RoboDK station: irb120.rdk

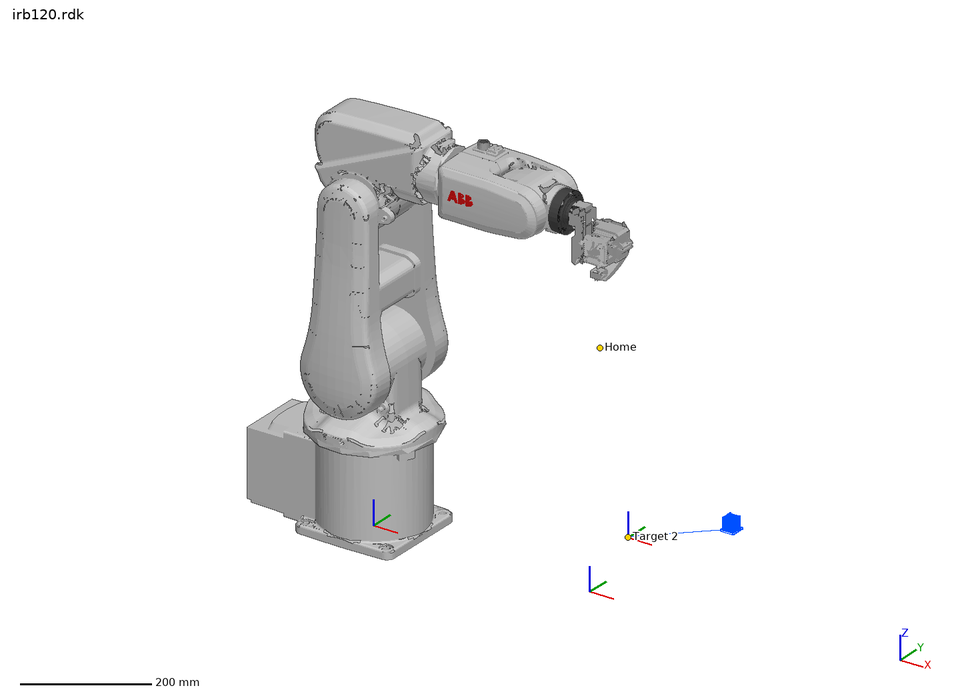
[picture v0: the station drawn from its stored meshes, robots at their saved joint values, targets as dots, program paths as lines]
Station irb120_V12 (saved by RoboDK 5.2.5). Poses are relative to the parent item; angles as X-Y-Z fixed-axis rotations.
  - frame ABB IRB 120-3/0.6 Base at (-494.33, 30.55, 0) mm
    - robot ABB IRB 120-3/0.6: 6 axes, payload 3 kg, reach 580 mm, repeatability 0.01 mm, weight 25 kg
        modified DH rows (alpha deg, a mm, theta deg, d mm): 0, 0, 0, 290; -90, 0, -90, 0; 0, 270, 0, 0; -90, 70, 0, 302; 90, 0, 0, 0; -90, 0, 180, 72
        joint limits [-165, -110, -90, -160, -120, -400] to [165, 110, 70, 160, 120, 400]; home [0, 0, 0, 0, 0, 0]; saved at [0, 0, 0, 0, 0, 0]
      - tool EndEffector, TCP at (101, 0, 38) mm, rotated rx 0 ry 90 rz 0 deg, size 98.6 x 123.3 x 80.9 mm, geometry from EndEffector.stl
  - frame Robot Table at (-94.33, 30.55, 0) mm
    - object Table at (0, 0, 0) mm, size 926 x 772 x 180 mm, geometry from Table.stl
  - frame Print at (40, -60, 165.5) mm
    - target Home (joint target) at (16.67, -99.45, 364) mm, rotated rx -180 ry 0 rz -180 deg; joints [0, 0, 0, 0, 0, 0] of ABB IRB 120-3/0.6
    - target Target 2 (Cartesian target) at (0, 0, 0) mm, rotated rx 180 ry 0 rz 180 deg; joints [-12.046, 47.993, 6.255, -14.732, -55.151, 8.545] of ABB IRB 120-3/0.6
  - Python program Prog2 (listed below)
  - camera Camera 1
  - frame Frame 4 at (1070.92, -4.45, 581.3) mm, rotated rx -103 ry 0 rz 90 deg
  - program out (41618 instructions, listed below)
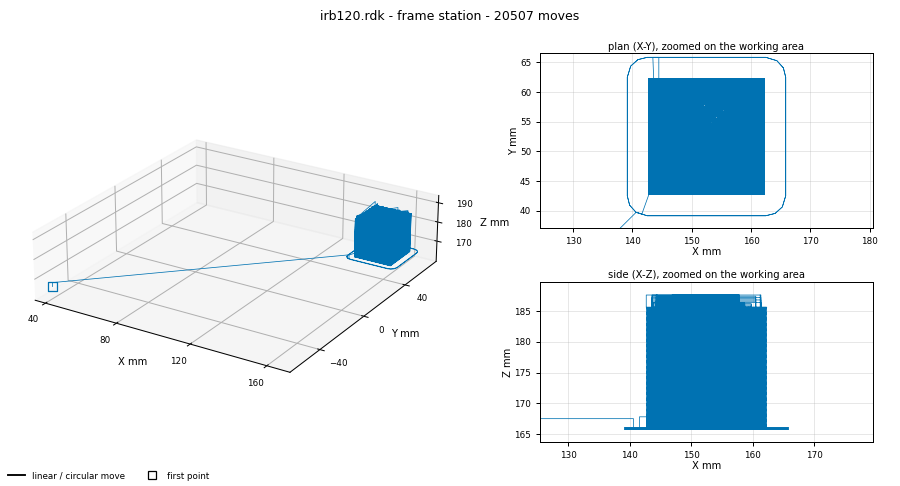
[picture p0: tool path of irb120.rdk in frame station, 20507 of 20507 moves have a stored position in this frame; points joined in program order, loops and branches not executed]

--- Python program Prog2 ---
# Type help("robolink") or help("robodk") for more information
# Press F5 to run the script
# Documentation: https://robodk.com/doc/en/RoboDK-API.html
# Reference:     https://robodk.com/doc/en/PythonAPI/index.html
# Note: It is not required to keep a copy of this file, your python script is saved with the station
from robolink import *    # RoboDK API
from robodk import *      # Robot toolbox
RDK = Robolink()
import cv2
import tempfile
import numpy as np
import math
# # Notify user:
# print('To edit this program:\nright click on the Python program, then, select "Edit Python script"')

# RDK = Robolink() # connect to the RoboDK API (RoboDK starts if it has not started)
# robot  = RDK.Item('', ITEM_TYPE_ROBOT)   # Retrieve the robot
# joints = robot.Joints().list()          # retrieve the current robot joints as a list
# joints[5] = 20                           # set joint 6 to 0 deg
# robot.MoveJ(joints)
# s=robot.JointPoses()
# Print("finish")
CAM_NAME = "Camera 1"
cam_item = RDK.Item(CAM_NAME, ITEM_TYPE_CAMERA)
if not cam_item.Valid():
    raise Exception("Camera not found! %s" % CAM_NAME)

tempdir = tempfile.gettempdir()
snapshot_file = tempdir + "\\sift_temp.png"
print(snapshot_file)
imgdir="C:/Users/dell/Desktop/RoboDk/Robotirb120/00006000.jpg"
image = cv2.imread(imgdir)
image=cv2.resize(image,(640,480))
while(1):
    RDK.Cam2D_Snapshot(snapshot_file, cam_item)
    img_scene = cv2.imread(snapshot_file, cv2.IMREAD_GRAYSCALE)
    img_scene=cv2.resize(img_scene,(640,480))
    (thresh, im_bw) = cv2.threshold(img_scene, 128, 255, cv2.THRESH_BINARY | cv2.THRESH_OTSU)
    # print(image.shape)
    # print(im_bw.shape)
    kernel = np.ones((3,3),np.uint8)
    closing = cv2.morphologyEx(im_bw, cv2.MORPH_CLOSE, kernel)
    gradient = cv2.morphologyEx(im_bw, cv2.MORPH_GRADIENT, kernel)
    masked = cv2.bitwise_and(image, image, mask=closing)
    vis = np.concatenate((image,masked), axis=1)
    cv2.imshow("image3",masked)
    key = cv2.waitKey(1)
    if key == 27:
        break  # User pressed ESC, exit

--- program out (robot ABB IRB 120-3/0.6) ---
  Set Ref.: Print
  Set Tool at (101, 0, 38) mm, rotated rx 0 ry 90 rz 0 deg
  Smooth(2)
  Set accel. (1000.0 mm/s2)
  Call Mcode M107
  MoveJ (T0) to (0, 0, 0) mm, rotated rx 180 ry 0 rz -180 deg; joints [0, 0, 0, 0, 0, 0]
  Call Mcode M190 S50
  MoveL (T1) to (0, 0, 0) mm, rotated rx 180 ry 0 rz -180 deg; joints [0, 0, 0, 0, 0, 0]
  Call Mcode M104 S200
  MoveL (T2) to (0, 0, 0) mm, rotated rx 180 ry 0 rz -180 deg; joints [0, 0, 0, 0, 0, 0]
  Call Mcode M109 S200
  MoveL (T3) to (0, 0, 0) mm, rotated rx 180 ry 0 rz -180 deg; joints [0, 0, 0, 0, 0, 0]
  Call Mcode M83
  MoveL (T4) to (0, 0, 0) mm, rotated rx 180 ry 0 rz -180 deg; joints [0, 0, 0, 0, 0, 0]
  Call Mcode M107
  MoveL (T5) to (0, 0, 0) mm, rotated rx 180 ry 0 rz -180 deg; joints [0, 0, 0, 0, 0, 0]
  Set speed (45.0 mm/s)
  Call Extruder -2.0
  MoveL (T6) to (0, 0, 0) mm, rotated rx 180 ry 0 rz -180 deg; joints [0, 0, 0, 0, 0, 0]
  Set speed (150.0 mm/s)
  MoveL (T7) to (0, 0, 2) mm, rotated rx 180 ry 0 rz -180 deg; joints [0, 0, 0, 0, 0, 0]
  MoveL (T8) to (100.63, 99.72, 2) mm, rotated rx 180 ry 0 rz -180 deg; joints [0, 0, 0, 0, 0, 0]
  MoveL (T9) to (100.63, 99.72, 0.3) mm, rotated rx 180 ry 0 rz -180 deg; joints [0, 0, 0, 0, 0, 0]
  Set speed (40.0 mm/s)
  Call Extruder 2.0
  MoveL (T10) to (100.63, 99.72, 0.3) mm, rotated rx 180 ry 0 rz -180 deg; joints [0, 0, 0, 0, 0, 0]
  Call Extruder 2.0
  Call Mcode M204 P1000
  MoveL (T11) to (100.63, 99.72, 0.3) mm, rotated rx 180 ry 0 rz -180 deg; joints [0, 0, 0, 0, 0, 0]
  Set speed (20.0 mm/s)
  MoveL (T12) to (100.63, 99.72, 0.3) mm, rotated rx 180 ry 0 rz -180 deg; joints [0, 0, 0, 0, 0, 0]
  Call Extruder 0.07812
  MoveL (T13) to (102.5, 99.14, 0.3) mm, rotated rx 180 ry 0 rz -180 deg; joints [0, 0, 0, 0, 0, 0]
  Call Extruder 0.79839
  MoveL (T14) to (122.5, 99.14, 0.3) mm, rotated rx 180 ry 0 rz -180 deg; joints [0, 0, 0, 0, 0, 0]
  Call Extruder 0.06492
  MoveL (T15) to (124.08, 99.54, 0.3) mm, rotated rx 180 ry 0 rz -180 deg; joints [0, 0, 0, 0, 0, 0]
  Call Extruder 0.06492
  MoveL (T16) to (125.28, 100.63, 0.3) mm, rotated rx 180 ry 0 rz -180 deg; joints [0, 0, 0, 0, 0, 0]
  Call Extruder 0.07812
  MoveL (T17) to (125.86, 102.5, 0.3) mm, rotated rx 180 ry 0 rz -180 deg; joints [0, 0, 0, 0, 0, 0]
  Call Extruder 0.79839
  MoveL (T18) to (125.86, 122.5, 0.3) mm, rotated rx 180 ry 0 rz -180 deg; joints [0, 0, 0, 0, 0, 0]
  Call Extruder 0.06492
  MoveL (T19) to (125.46, 124.08, 0.3) mm, rotated rx 180 ry 0 rz -180 deg; joints [0, 0, 0, 0, 0, 0]
  Call Extruder 0.06492
  MoveL (T20) to (124.37, 125.28, 0.3) mm, rotated rx 180 ry 0 rz -180 deg; joints [0, 0, 0, 0, 0, 0]
  Call Extruder 0.07812
  MoveL (T21) to (122.5, 125.86, 0.3) mm, rotated rx 180 ry 0 rz -180 deg; joints [0, 0, 0, 0, 0, 0]
  Call Extruder 0.79839
  MoveL (T22) to (102.5, 125.86, 0.3) mm, rotated rx 180 ry 0 rz -180 deg; joints [0, 0, 0, 0, 0, 0]
  Call Extruder 0.06492
  MoveL (T23) to (100.92, 125.46, 0.3) mm, rotated rx 180 ry 0 rz -180 deg; joints [0, 0, 0, 0, 0, 0]
  Call Extruder 0.06492
  MoveL (T24) to (99.72, 124.37, 0.3) mm, rotated rx 180 ry 0 rz -180 deg; joints [0, 0, 0, 0, 0, 0]
  Call Extruder 0.07812
  MoveL (T25) to (99.14, 122.5, 0.3) mm, rotated rx 180 ry 0 rz -180 deg; joints [0, 0, 0, 0, 0, 0]
  Call Extruder 0.79839
  MoveL (T26) to (99.14, 102.5, 0.3) mm, rotated rx 180 ry 0 rz -180 deg; joints [0, 0, 0, 0, 0, 0]
  Call Extruder 0.06492
  MoveL (T27) to (99.54, 100.92, 0.3) mm, rotated rx 180 ry 0 rz -180 deg; joints [0, 0, 0, 0, 0, 0]
  Call Extruder 0.06252
  MoveL (T28) to (100.59, 99.76, 0.3) mm, rotated rx 180 ry 0 rz -180 deg; joints [0, 0, 0, 0, 0, 0]
  Set speed (45.0 mm/s)
  Call Extruder -1.6
  MoveL (T29) to (100.59, 99.76, 0.3) mm, rotated rx 180 ry 0 rz -180 deg; joints [0, 0, 0, 0, 0, 0]
  Set speed (120.0 mm/s)
  MoveL (T30) to (100.59, 99.76, 0.3) mm, rotated rx 180 ry 0 rz -180 deg; joints [0, 0, 0, 0, 0, 0]
  Call Extruder -0.38
  MoveL (T31) to (101.6, 99.43, 0.3) mm, rotated rx 180 ry 0 rz -180 deg; joints [0, 0, 0, 0, 0, 0]
  Set speed (45.0 mm/s)
  Call Extruder -0.02
  MoveL (T32) to (101.6, 99.43, 0.3) mm, rotated rx 180 ry 0 rz -180 deg; joints [0, 0, 0, 0, 0, 0]
  Set speed (150.0 mm/s)
  MoveL (T33) to (101.6, 99.43, 2.3) mm, rotated rx 180 ry 0 rz -180 deg; joints [0, 0, 0, 0, 0, 0]
  MoveL (T34) to (102.81, 102.81, 2.3) mm, rotated rx 180 ry 0 rz -180 deg; joints [0, 0, 0, 0, 0, 0]
  MoveL (T35) to (102.81, 102.81, 0.3) mm, rotated rx 180 ry 0 rz -180 deg; joints [0, 0, 0, 0, 0, 0]
  Set speed (40.0 mm/s)
  Call Extruder 2.0
  MoveL (T36) to (102.81, 102.81, 0.3) mm, rotated rx 180 ry 0 rz -180 deg; joints [0, 0, 0, 0, 0, 0]
  Set speed (20.0 mm/s)
  MoveL (T37) to (102.81, 102.81, 0.3) mm, rotated rx 180 ry 0 rz -180 deg; joints [0, 0, 0, 0, 0, 0]
  Call Extruder 0.77364
  MoveL (T38) to (122.19, 102.81, 0.3) mm, rotated rx 180 ry 0 rz -180 deg; joints [0, 0, 0, 0, 0, 0]
  Call Extruder 0.77364
  MoveL (T39) to (122.19, 122.19, 0.3) mm, rotated rx 180 ry 0 rz -180 deg; joints [0, 0, 0, 0, 0, 0]
  Call Extruder 0.77364
  MoveL (T40) to (102.81, 122.19, 0.3) mm, rotated rx 180 ry 0 rz -180 deg; joints [0, 0, 0, 0, 0, 0]
  Call Extruder 0.77124
  MoveL (T41) to (102.81, 102.87, 0.3) mm, rotated rx 180 ry 0 rz -180 deg; joints [0, 0, 0, 0, 0, 0]
  Set speed (150.0 mm/s)
  MoveL (T42) to (103.2, 102.91, 0.3) mm, rotated rx 180 ry 0 rz -180 deg; joints [0, 0, 0, 0, 0, 0]
  Set speed (45.0 mm/s)
  Call Extruder -1.6
  MoveL (T43) to (103.2, 102.91, 0.3) mm, rotated rx 180 ry 0 rz -180 deg; joints [0, 0, 0, 0, 0, 0]
  Set speed (120.0 mm/s)
  MoveL (T44) to (103.2, 102.91, 0.3) mm, rotated rx 180 ry 0 rz -180 deg; joints [0, 0, 0, 0, 0, 0]
  Call Extruder -0.38
  MoveL (T45) to (103.88, 102.87, 0.3) mm, rotated rx 180 ry 0 rz -180 deg; joints [0, 0, 0, 0, 0, 0]
  Set speed (45.0 mm/s)
  Call Extruder -0.02
  MoveL (T46) to (103.88, 102.87, 0.3) mm, rotated rx 180 ry 0 rz -180 deg; joints [0, 0, 0, 0, 0, 0]
  Set speed (150.0 mm/s)
  MoveL (T47) to (103.88, 102.87, 2.3) mm, rotated rx 180 ry 0 rz -180 deg; joints [0, 0, 0, 0, 0, 0]
  MoveL (T48) to (121.83, 121.83, 2.3) mm, rotated rx 180 ry 0 rz -180 deg; joints [0, 0, 0, 0, 0, 0]
  MoveL (T49) to (121.83, 121.83, 0.3) mm, rotated rx 180 ry 0 rz -180 deg; joints [0, 0, 0, 0, 0, 0]
  Set speed (40.0 mm/s)
  Call Extruder 2.0
  MoveL (T50) to (121.83, 121.83, 0.3) mm, rotated rx 180 ry 0 rz -180 deg; joints [0, 0, 0, 0, 0, 0]
  Set speed (20.0 mm/s)
  MoveL (T51) to (121.83, 121.83, 0.3) mm, rotated rx 180 ry 0 rz -180 deg; joints [0, 0, 0, 0, 0, 0]
  Call Extruder 0.74524
  MoveL (T52) to (103.17, 121.83, 0.3) mm, rotated rx 180 ry 0 rz -180 deg; joints [0, 0, 0, 0, 0, 0]
  Call Extruder 0.74524
  MoveL (T53) to (103.17, 103.17, 0.3) mm, rotated rx 180 ry 0 rz -180 deg; joints [0, 0, 0, 0, 0, 0]
  Call Extruder 0.74524
  MoveL (T54) to (121.83, 103.17, 0.3) mm, rotated rx 180 ry 0 rz -180 deg; joints [0, 0, 0, 0, 0, 0]
  Call Extruder 0.74285
  MoveL (T55) to (121.83, 121.77, 0.3) mm, rotated rx 180 ry 0 rz -180 deg; joints [0, 0, 0, 0, 0, 0]
  Set speed (150.0 mm/s)
  MoveL (T56) to (121.48, 121.48, 0.3) mm, rotated rx 180 ry 0 rz -180 deg; joints [0, 0, 0, 0, 0, 0]
  Set speed (20.0 mm/s)
  MoveL (T57) to (121.48, 121.48, 0.3) mm, rotated rx 180 ry 0 rz -180 deg; joints [0, 0, 0, 0, 0, 0]
  Call Extruder 0.71685
  MoveL (T58) to (103.52, 121.48, 0.3) mm, rotated rx 180 ry 0 rz -180 deg; joints [0, 0, 0, 0, 0, 0]
  Call Extruder 0.71685
  MoveL (T59) to (103.52, 103.52, 0.3) mm, rotated rx 180 ry 0 rz -180 deg; joints [0, 0, 0, 0, 0, 0]
  Call Extruder 0.71685
  MoveL (T60) to (121.48, 103.52, 0.3) mm, rotated rx 180 ry 0 rz -180 deg; joints [0, 0, 0, 0, 0, 0]
  Call Extruder 0.71446
  MoveL (T61) to (121.48, 121.42, 0.3) mm, rotated rx 180 ry 0 rz -180 deg; joints [0, 0, 0, 0, 0, 0]
  Set speed (45.0 mm/s)
  Call Extruder -1.6
  MoveL (T62) to (121.48, 121.42, 0.3) mm, rotated rx 180 ry 0 rz -180 deg; joints [0, 0, 0, 0, 0, 0]
  Set speed (120.0 mm/s)
  MoveL (T63) to (121.48, 121.42, 0.3) mm, rotated rx 180 ry 0 rz -180 deg; joints [0, 0, 0, 0, 0, 0]
  Call Extruder -0.38
  MoveL (T64) to (120.41, 121.42, 0.3) mm, rotated rx 180 ry 0 rz -180 deg; joints [0, 0, 0, 0, 0, 0]
  Set speed (45.0 mm/s)
  Call Extruder -0.02
  MoveL (T65) to (120.41, 121.42, 0.3) mm, rotated rx 180 ry 0 rz -180 deg; joints [0, 0, 0, 0, 0, 0]
  Set speed (150.0 mm/s)
  MoveL (T66) to (120.41, 121.42, 2.3) mm, rotated rx 180 ry 0 rz -180 deg; joints [0, 0, 0, 0, 0, 0]
  MoveL (T67) to (120.65, 103.63, 2.3) mm, rotated rx 180 ry 0 rz -180 deg; joints [0, 0, 0, 0, 0, 0]
  MoveL (T68) to (120.65, 103.63, 0.3) mm, rotated rx 180 ry 0 rz -180 deg; joints [0, 0, 0, 0, 0, 0]
  Set speed (40.0 mm/s)
  Call Extruder 2.0
  MoveL (T69) to (120.65, 103.63, 0.3) mm, rotated rx 180 ry 0 rz -180 deg; joints [0, 0, 0, 0, 0, 0]
  Set speed (20.0 mm/s)
  MoveL (T70) to (120.65, 103.63, 0.3) mm, rotated rx 180 ry 0 rz -180 deg; joints [0, 0, 0, 0, 0, 0]
  Call Extruder 0.0323
  MoveL (T71) to (121.21, 104.19, 0.3) mm, rotated rx 180 ry 0 rz -180 deg; joints [0, 0, 0, 0, 0, 0]
  Call Extruder 0.02048
  MoveL (T72) to (121.21, 104.7, 0.3) mm, rotated rx 180 ry 0 rz -180 deg; joints [0, 0, 0, 0, 0, 0]
  Call Extruder 0.05214
  MoveL (T73) to (120.3, 103.79, 0.3) mm, rotated rx 180 ry 0 rz -180 deg; joints [0, 0, 0, 0, 0, 0]
  Call Extruder 0.02048
  MoveL (T74) to (119.79, 103.79, 0.3) mm, rotated rx 180 ry 0 rz -180 deg; joints [0, 0, 0, 0, 0, 0]
  Call Extruder 0.08111
  MoveL (T75) to (121.21, 105.21, 0.3) mm, rotated rx 180 ry 0 rz -180 deg; joints [0, 0, 0, 0, 0, 0]
  Call Extruder 0.02048
  MoveL (T76) to (121.21, 105.72, 0.3) mm, rotated rx 180 ry 0 rz -180 deg; joints [0, 0, 0, 0, 0, 0]
  Call Extruder 0.11008
  MoveL (T77) to (119.28, 103.79, 0.3) mm, rotated rx 180 ry 0 rz -180 deg; joints [0, 0, 0, 0, 0, 0]
  Call Extruder 0.02048
  MoveL (T78) to (118.77, 103.79, 0.3) mm, rotated rx 180 ry 0 rz -180 deg; joints [0, 0, 0, 0, 0, 0]
  Call Extruder 0.13905
  MoveL (T79) to (121.21, 106.23, 0.3) mm, rotated rx 180 ry 0 rz -180 deg; joints [0, 0, 0, 0, 0, 0]
  Call Extruder 0.02048
  MoveL (T80) to (121.21, 106.73, 0.3) mm, rotated rx 180 ry 0 rz -180 deg; joints [0, 0, 0, 0, 0, 0]
  Call Extruder 0.16801
  MoveL (T81) to (118.27, 103.79, 0.3) mm, rotated rx 180 ry 0 rz -180 deg; joints [0, 0, 0, 0, 0, 0]
  Call Extruder 0.02048
  MoveL (T82) to (117.76, 103.79, 0.3) mm, rotated rx 180 ry 0 rz -180 deg; joints [0, 0, 0, 0, 0, 0]
  Call Extruder 0.19698
  MoveL (T83) to (121.21, 107.24, 0.3) mm, rotated rx 180 ry 0 rz -180 deg; joints [0, 0, 0, 0, 0, 0]
  Call Extruder 0.02048
  MoveL (T84) to (121.21, 107.75, 0.3) mm, rotated rx 180 ry 0 rz -180 deg; joints [0, 0, 0, 0, 0, 0]
  Call Extruder 0.22595
  MoveL (T85) to (117.25, 103.79, 0.3) mm, rotated rx 180 ry 0 rz -180 deg; joints [0, 0, 0, 0, 0, 0]
  Call Extruder 0.02048
  MoveL (T86) to (116.74, 103.79, 0.3) mm, rotated rx 180 ry 0 rz -180 deg; joints [0, 0, 0, 0, 0, 0]
  Call Extruder 0.25492
  MoveL (T87) to (121.21, 108.26, 0.3) mm, rotated rx 180 ry 0 rz -180 deg; joints [0, 0, 0, 0, 0, 0]
  Call Extruder 0.02048
  MoveL (T88) to (121.21, 108.77, 0.3) mm, rotated rx 180 ry 0 rz -180 deg; joints [0, 0, 0, 0, 0, 0]
  Call Extruder 0.28388
  MoveL (T89) to (116.23, 103.79, 0.3) mm, rotated rx 180 ry 0 rz -180 deg; joints [0, 0, 0, 0, 0, 0]
  Call Extruder 0.02048
  MoveL (T90) to (115.73, 103.79, 0.3) mm, rotated rx 180 ry 0 rz -180 deg; joints [0, 0, 0, 0, 0, 0]
  Call Extruder 0.31285
  MoveL (T91) to (121.21, 109.27, 0.3) mm, rotated rx 180 ry 0 rz -180 deg; joints [0, 0, 0, 0, 0, 0]
  Call Extruder 0.02048
  MoveL (T92) to (121.21, 109.78, 0.3) mm, rotated rx 180 ry 0 rz -180 deg; joints [0, 0, 0, 0, 0, 0]
  Call Extruder 0.34182
  MoveL (T93) to (115.22, 103.79, 0.3) mm, rotated rx 180 ry 0 rz -180 deg; joints [0, 0, 0, 0, 0, 0]
  Call Extruder 0.02048
  MoveL (T94) to (114.71, 103.79, 0.3) mm, rotated rx 180 ry 0 rz -180 deg; joints [0, 0, 0, 0, 0, 0]
  Call Extruder 0.37079
  MoveL (T95) to (121.21, 110.29, 0.3) mm, rotated rx 180 ry 0 rz -180 deg; joints [0, 0, 0, 0, 0, 0]
  Call Extruder 0.02048
  MoveL (T96) to (121.21, 110.8, 0.3) mm, rotated rx 180 ry 0 rz -180 deg; joints [0, 0, 0, 0, 0, 0]
  Call Extruder 0.39975
  MoveL (T97) to (114.2, 103.79, 0.3) mm, rotated rx 180 ry 0 rz -180 deg; joints [0, 0, 0, 0, 0, 0]
  Call Extruder 0.02048
  MoveL (T98) to (113.69, 103.79, 0.3) mm, rotated rx 180 ry 0 rz -180 deg; joints [0, 0, 0, 0, 0, 0]
  Call Extruder 0.42872
  MoveL (T99) to (121.21, 111.31, 0.3) mm, rotated rx 180 ry 0 rz -180 deg; joints [0, 0, 0, 0, 0, 0]
  Call Extruder 0.02048
  MoveL (T100) to (121.21, 111.81, 0.3) mm, rotated rx 180 ry 0 rz -180 deg; joints [0, 0, 0, 0, 0, 0]
  Call Extruder 0.45769
  MoveL (T101) to (113.19, 103.79, 0.3) mm, rotated rx 180 ry 0 rz -180 deg; joints [0, 0, 0, 0, 0, 0]
  Call Extruder 0.02048
  MoveL (T102) to (112.68, 103.79, 0.3) mm, rotated rx 180 ry 0 rz -180 deg; joints [0, 0, 0, 0, 0, 0]
  Call Extruder 0.48666
  MoveL (T103) to (121.21, 112.32, 0.3) mm, rotated rx 180 ry 0 rz -180 deg; joints [0, 0, 0, 0, 0, 0]
  Call Extruder 0.02048
  MoveL (T104) to (121.21, 112.83, 0.3) mm, rotated rx 180 ry 0 rz -180 deg; joints [0, 0, 0, 0, 0, 0]
  Call Extruder 0.51562
  MoveL (T105) to (112.17, 103.79, 0.3) mm, rotated rx 180 ry 0 rz -180 deg; joints [0, 0, 0, 0, 0, 0]
  Call Extruder 0.02048
  MoveL (T106) to (111.66, 103.79, 0.3) mm, rotated rx 180 ry 0 rz -180 deg; joints [0, 0, 0, 0, 0, 0]
  Call Extruder 0.54459
  MoveL (T107) to (121.21, 113.34, 0.3) mm, rotated rx 180 ry 0 rz -180 deg; joints [0, 0, 0, 0, 0, 0]
  Call Extruder 0.02048
  MoveL (T108) to (121.21, 113.85, 0.3) mm, rotated rx 180 ry 0 rz -180 deg; joints [0, 0, 0, 0, 0, 0]
  Call Extruder 0.57356
  MoveL (T109) to (111.15, 103.79, 0.3) mm, rotated rx 180 ry 0 rz -180 deg; joints [0, 0, 0, 0, 0, 0]
  Call Extruder 0.02048
  MoveL (T110) to (110.65, 103.79, 0.3) mm, rotated rx 180 ry 0 rz -180 deg; joints [0, 0, 0, 0, 0, 0]
  Call Extruder 0.60253
  MoveL (T111) to (121.21, 114.35, 0.3) mm, rotated rx 180 ry 0 rz -180 deg; joints [0, 0, 0, 0, 0, 0]
  Call Extruder 0.02048
  MoveL (T112) to (121.21, 114.86, 0.3) mm, rotated rx 180 ry 0 rz -180 deg; joints [0, 0, 0, 0, 0, 0]
  Call Extruder 0.63149
  MoveL (T113) to (110.14, 103.79, 0.3) mm, rotated rx 180 ry 0 rz -180 deg; joints [0, 0, 0, 0, 0, 0]
  Call Extruder 0.02048
  MoveL (T114) to (109.63, 103.79, 0.3) mm, rotated rx 180 ry 0 rz -180 deg; joints [0, 0, 0, 0, 0, 0]
  Call Extruder 0.66046
  MoveL (T115) to (121.21, 115.37, 0.3) mm, rotated rx 180 ry 0 rz -180 deg; joints [0, 0, 0, 0, 0, 0]
  Call Extruder 0.02048
  MoveL (T116) to (121.21, 115.88, 0.3) mm, rotated rx 180 ry 0 rz -180 deg; joints [0, 0, 0, 0, 0, 0]
  Call Extruder 0.68943
  MoveL (T117) to (109.12, 103.79, 0.3) mm, rotated rx 180 ry 0 rz -180 deg; joints [0, 0, 0, 0, 0, 0]
  Call Extruder 0.02048
  MoveL (T118) to (108.61, 103.79, 0.3) mm, rotated rx 180 ry 0 rz -180 deg; joints [0, 0, 0, 0, 0, 0]
  Call Extruder 0.7184
  MoveL (T119) to (121.21, 116.39, 0.3) mm, rotated rx 180 ry 0 rz -180 deg; joints [0, 0, 0, 0, 0, 0]
  Call Extruder 0.02048
  MoveL (T120) to (121.21, 116.89, 0.3) mm, rotated rx 180 ry 0 rz -180 deg; joints [0, 0, 0, 0, 0, 0]
  Call Extruder 0.74736
  MoveL (T121) to (108.11, 103.79, 0.3) mm, rotated rx 180 ry 0 rz -180 deg; joints [0, 0, 0, 0, 0, 0]
  Call Extruder 0.02048
  MoveL (T122) to (107.6, 103.79, 0.3) mm, rotated rx 180 ry 0 rz -180 deg; joints [0, 0, 0, 0, 0, 0]
  Call Extruder 0.77633
  MoveL (T123) to (121.21, 117.4, 0.3) mm, rotated rx 180 ry 0 rz -180 deg; joints [0, 0, 0, 0, 0, 0]
  Call Extruder 0.02048
  MoveL (T124) to (121.21, 117.91, 0.3) mm, rotated rx 180 ry 0 rz -180 deg; joints [0, 0, 0, 0, 0, 0]
  Call Extruder 0.8053
  MoveL (T125) to (107.09, 103.79, 0.3) mm, rotated rx 180 ry 0 rz -180 deg; joints [0, 0, 0, 0, 0, 0]
  Call Extruder 0.02048
  MoveL (T126) to (106.58, 103.79, 0.3) mm, rotated rx 180 ry 0 rz -180 deg; joints [0, 0, 0, 0, 0, 0]
  Call Extruder 0.83426
  MoveL (T127) to (121.21, 118.42, 0.3) mm, rotated rx 180 ry 0 rz -180 deg; joints [0, 0, 0, 0, 0, 0]
  Call Extruder 0.02048
  MoveL (T128) to (121.21, 118.93, 0.3) mm, rotated rx 180 ry 0 rz -180 deg; joints [0, 0, 0, 0, 0, 0]
  Call Extruder 0.86323
  MoveL (T129) to (106.07, 103.79, 0.3) mm, rotated rx 180 ry 0 rz -180 deg; joints [0, 0, 0, 0, 0, 0]
  Call Extruder 0.02048
  MoveL (T130) to (105.57, 103.79, 0.3) mm, rotated rx 180 ry 0 rz -180 deg; joints [0, 0, 0, 0, 0, 0]
  Call Extruder 0.8922
  MoveL (T131) to (121.21, 119.43, 0.3) mm, rotated rx 180 ry 0 rz -180 deg; joints [0, 0, 0, 0, 0, 0]
  Call Extruder 0.02048
  MoveL (T132) to (121.21, 119.94, 0.3) mm, rotated rx 180 ry 0 rz -180 deg; joints [0, 0, 0, 0, 0, 0]
  Call Extruder 0.92117
  MoveL (T133) to (105.06, 103.79, 0.3) mm, rotated rx 180 ry 0 rz -180 deg; joints [0, 0, 0, 0, 0, 0]
  Call Extruder 0.02048
  MoveL (T134) to (104.55, 103.79, 0.3) mm, rotated rx 180 ry 0 rz -180 deg; joints [0, 0, 0, 0, 0, 0]
  Call Extruder 0.95013
  MoveL (T135) to (121.21, 120.45, 0.3) mm, rotated rx 180 ry 0 rz -180 deg; joints [0, 0, 0, 0, 0, 0]
  Call Extruder 0.02048
  MoveL (T136) to (121.21, 120.96, 0.3) mm, rotated rx 180 ry 0 rz -180 deg; joints [0, 0, 0, 0, 0, 0]
  Call Extruder 0.9791
  MoveL (T137) to (104.04, 103.79, 0.3) mm, rotated rx 180 ry 0 rz -180 deg; joints [0, 0, 0, 0, 0, 0]
  Call Extruder 0.01024
  MoveL (T138) to (103.79, 103.79, 0.3) mm, rotated rx 180 ry 0 rz -180 deg; joints [0, 0, 0, 0, 0, 0]
  Call Extruder 0.01024
  MoveL (T139) to (103.79, 104.04, 0.3) mm, rotated rx 180 ry 0 rz -180 deg; joints [0, 0, 0, 0, 0, 0]
  Call Extruder 0.9791
  MoveL (T140) to (120.96, 121.21, 0.3) mm, rotated rx 180 ry 0 rz -180 deg; joints [0, 0, 0, 0, 0, 0]
  Call Extruder 0.02048
  MoveL (T141) to (120.45, 121.21, 0.3) mm, rotated rx 180 ry 0 rz -180 deg; joints [0, 0, 0, 0, 0, 0]
  Call Extruder 0.95013
  MoveL (T142) to (103.79, 104.55, 0.3) mm, rotated rx 180 ry 0 rz -180 deg; joints [0, 0, 0, 0, 0, 0]
  Call Extruder 0.02048
  MoveL (T143) to (103.79, 105.06, 0.3) mm, rotated rx 180 ry 0 rz -180 deg; joints [0, 0, 0, 0, 0, 0]
  Call Extruder 0.92116
  MoveL (T144) to (119.94, 121.21, 0.3) mm, rotated rx 180 ry 0 rz -180 deg; joints [0, 0, 0, 0, 0, 0]
  Call Extruder 0.02048
  MoveL (T145) to (119.43, 121.21, 0.3) mm, rotated rx 180 ry 0 rz -180 deg; joints [0, 0, 0, 0, 0, 0]
  Call Extruder 0.8922
  MoveL (T146) to (103.79, 105.57, 0.3) mm, rotated rx 180 ry 0 rz -180 deg; joints [0, 0, 0, 0, 0, 0]
  Call Extruder 0.02048
  MoveL (T147) to (103.79, 106.07, 0.3) mm, rotated rx 180 ry 0 rz -180 deg; joints [0, 0, 0, 0, 0, 0]
  Call Extruder 0.86323
  MoveL (T148) to (118.93, 121.21, 0.3) mm, rotated rx 180 ry 0 rz -180 deg; joints [0, 0, 0, 0, 0, 0]
  Call Extruder 0.02048
  MoveL (T149) to (118.42, 121.21, 0.3) mm, rotated rx 180 ry 0 rz -180 deg; joints [0, 0, 0, 0, 0, 0]
  Call Extruder 0.83426
  MoveL (T150) to (103.79, 106.58, 0.3) mm, rotated rx 180 ry 0 rz -180 deg; joints [0, 0, 0, 0, 0, 0]
  Call Extruder 0.02048
  MoveL (T151) to (103.79, 107.09, 0.3) mm, rotated rx 180 ry 0 rz -180 deg; joints [0, 0, 0, 0, 0, 0]
  Call Extruder 0.80529
  MoveL (T152) to (117.91, 121.21, 0.3) mm, rotated rx 180 ry 0 rz -180 deg; joints [0, 0, 0, 0, 0, 0]
  Call Extruder 0.02048
  MoveL (T153) to (117.4, 121.21, 0.3) mm, rotated rx 180 ry 0 rz -180 deg; joints [0, 0, 0, 0, 0, 0]
  Call Extruder 0.77633
  MoveL (T154) to (103.79, 107.6, 0.3) mm, rotated rx 180 ry 0 rz -180 deg; joints [0, 0, 0, 0, 0, 0]
  Call Extruder 0.02048
  MoveL (T155) to (103.79, 108.11, 0.3) mm, rotated rx 180 ry 0 rz -180 deg; joints [0, 0, 0, 0, 0, 0]
  Call Extruder 0.74736
  MoveL (T156) to (116.89, 121.21, 0.3) mm, rotated rx 180 ry 0 rz -180 deg; joints [0, 0, 0, 0, 0, 0]
  Call Extruder 0.02048
  MoveL (T157) to (116.39, 121.21, 0.3) mm, rotated rx 180 ry 0 rz -180 deg; joints [0, 0, 0, 0, 0, 0]
  Call Extruder 0.71839
  MoveL (T158) to (103.79, 108.61, 0.3) mm, rotated rx 180 ry 0 rz -180 deg; joints [0, 0, 0, 0, 0, 0]
  Call Extruder 0.02048
  MoveL (T159) to (103.79, 109.12, 0.3) mm, rotated rx 180 ry 0 rz -180 deg; joints [0, 0, 0, 0, 0, 0]
  Call Extruder 0.68942
  MoveL (T160) to (115.88, 121.21, 0.3) mm, rotated rx 180 ry 0 rz -180 deg; joints [0, 0, 0, 0, 0, 0]
  Call Extruder 0.02048
  MoveL (T161) to (115.37, 121.21, 0.3) mm, rotated rx 180 ry 0 rz -180 deg; joints [0, 0, 0, 0, 0, 0]
  Call Extruder 0.66046
  MoveL (T162) to (103.79, 109.63, 0.3) mm, rotated rx 180 ry 0 rz -180 deg; joints [0, 0, 0, 0, 0, 0]
  Call Extruder 0.02048
  MoveL (T163) to (103.79, 110.14, 0.3) mm, rotated rx 180 ry 0 rz -180 deg; joints [0, 0, 0, 0, 0, 0]
  Call Extruder 0.63149
  MoveL (T164) to (114.86, 121.21, 0.3) mm, rotated rx 180 ry 0 rz -180 deg; joints [0, 0, 0, 0, 0, 0]
  Call Extruder 0.02048
  MoveL (T165) to (114.35, 121.21, 0.3) mm, rotated rx 180 ry 0 rz -180 deg; joints [0, 0, 0, 0, 0, 0]
  Call Extruder 0.60252
  MoveL (T166) to (103.79, 110.65, 0.3) mm, rotated rx 180 ry 0 rz -180 deg; joints [0, 0, 0, 0, 0, 0]
  Call Extruder 0.02048
  MoveL (T167) to (103.79, 111.15, 0.3) mm, rotated rx 180 ry 0 rz -180 deg; joints [0, 0, 0, 0, 0, 0]
  Call Extruder 0.57356
  MoveL (T168) to (113.85, 121.21, 0.3) mm, rotated rx 180 ry 0 rz -180 deg; joints [0, 0, 0, 0, 0, 0]
  Call Extruder 0.02048
  MoveL (T169) to (113.34, 121.21, 0.3) mm, rotated rx 180 ry 0 rz -180 deg; joints [0, 0, 0, 0, 0, 0]
  Call Extruder 0.54459
  MoveL (T170) to (103.79, 111.66, 0.3) mm, rotated rx 180 ry 0 rz -180 deg; joints [0, 0, 0, 0, 0, 0]
  Call Extruder 0.02048
  MoveL (T171) to (103.79, 112.17, 0.3) mm, rotated rx 180 ry 0 rz -180 deg; joints [0, 0, 0, 0, 0, 0]
  Call Extruder 0.51562
  MoveL (T172) to (112.83, 121.21, 0.3) mm, rotated rx 180 ry 0 rz -180 deg; joints [0, 0, 0, 0, 0, 0]
  Call Extruder 0.02048
  MoveL (T173) to (112.32, 121.21, 0.3) mm, rotated rx 180 ry 0 rz -180 deg; joints [0, 0, 0, 0, 0, 0]
  Call Extruder 0.48665
  MoveL (T174) to (103.79, 112.68, 0.3) mm, rotated rx 180 ry 0 rz -180 deg; joints [0, 0, 0, 0, 0, 0]
  Call Extruder 0.02048
  MoveL (T175) to (103.79, 113.19, 0.3) mm, rotated rx 180 ry 0 rz -180 deg; joints [0, 0, 0, 0, 0, 0]
  Call Extruder 0.45769
  MoveL (T176) to (111.81, 121.21, 0.3) mm, rotated rx 180 ry 0 rz -180 deg; joints [0, 0, 0, 0, 0, 0]
  Call Extruder 0.02048
  MoveL (T177) to (111.31, 121.21, 0.3) mm, rotated rx 180 ry 0 rz -180 deg; joints [0, 0, 0, 0, 0, 0]
  Call Extruder 0.42872
  MoveL (T178) to (103.79, 113.69, 0.3) mm, rotated rx 180 ry 0 rz -180 deg; joints [0, 0, 0, 0, 0, 0]
  Call Extruder 0.02048
  MoveL (T179) to (103.79, 114.2, 0.3) mm, rotated rx 180 ry 0 rz -180 deg; joints [0, 0, 0, 0, 0, 0]
  Call Extruder 0.39975
  MoveL (T180) to (110.8, 121.21, 0.3) mm, rotated rx 180 ry 0 rz -180 deg; joints [0, 0, 0, 0, 0, 0]
  Call Extruder 0.02048
  MoveL (T181) to (110.29, 121.21, 0.3) mm, rotated rx 180 ry 0 rz -180 deg; joints [0, 0, 0, 0, 0, 0]
  Call Extruder 0.37078
  MoveL (T182) to (103.79, 114.71, 0.3) mm, rotated rx 180 ry 0 rz -180 deg; joints [0, 0, 0, 0, 0, 0]
  Call Extruder 0.02048
  MoveL (T183) to (103.79, 115.22, 0.3) mm, rotated rx 180 ry 0 rz -180 deg; joints [0, 0, 0, 0, 0, 0]
  Call Extruder 0.34182
  MoveL (T184) to (109.78, 121.21, 0.3) mm, rotated rx 180 ry 0 rz -180 deg; joints [0, 0, 0, 0, 0, 0]
  Call Extruder 0.02048
  MoveL (T185) to (109.27, 121.21, 0.3) mm, rotated rx 180 ry 0 rz -180 deg; joints [0, 0, 0, 0, 0, 0]
  Call Extruder 0.31285
  MoveL (T186) to (103.79, 115.73, 0.3) mm, rotated rx 180 ry 0 rz -180 deg; joints [0, 0, 0, 0, 0, 0]
  Call Extruder 0.02048
  MoveL (T187) to (103.79, 116.23, 0.3) mm, rotated rx 180 ry 0 rz -180 deg; joints [0, 0, 0, 0, 0, 0]
  Call Extruder 0.28388
  MoveL (T188) to (108.77, 121.21, 0.3) mm, rotated rx 180 ry 0 rz -180 deg; joints [0, 0, 0, 0, 0, 0]
  Call Extruder 0.02048
  MoveL (T189) to (108.26, 121.21, 0.3) mm, rotated rx 180 ry 0 rz -180 deg; joints [0, 0, 0, 0, 0, 0]
  Call Extruder 0.25491
  MoveL (T190) to (103.79, 116.74, 0.3) mm, rotated rx 180 ry 0 rz -180 deg; joints [0, 0, 0, 0, 0, 0]
  Call Extruder 0.02048
  MoveL (T191) to (103.79, 117.25, 0.3) mm, rotated rx 180 ry 0 rz -180 deg; joints [0, 0, 0, 0, 0, 0]
  Call Extruder 0.22595
  MoveL (T192) to (107.75, 121.21, 0.3) mm, rotated rx 180 ry 0 rz -180 deg; joints [0, 0, 0, 0, 0, 0]
  Call Extruder 0.02048
  MoveL (T193) to (107.24, 121.21, 0.3) mm, rotated rx 180 ry 0 rz -180 deg; joints [0, 0, 0, 0, 0, 0]
  Call Extruder 0.19698
  MoveL (T194) to (103.79, 117.76, 0.3) mm, rotated rx 180 ry 0 rz -180 deg; joints [0, 0, 0, 0, 0, 0]
  Call Extruder 0.02048
  MoveL (T195) to (103.79, 118.27, 0.3) mm, rotated rx 180 ry 0 rz -180 deg; joints [0, 0, 0, 0, 0, 0]
  Call Extruder 0.16801
  MoveL (T196) to (106.73, 121.21, 0.3) mm, rotated rx 180 ry 0 rz -180 deg; joints [0, 0, 0, 0, 0, 0]
  Call Extruder 0.02048
  MoveL (T197) to (106.23, 121.21, 0.3) mm, rotated rx 180 ry 0 rz -180 deg; joints [0, 0, 0, 0, 0, 0]
  Call Extruder 0.13904
  MoveL (T198) to (103.79, 118.77, 0.3) mm, rotated rx 180 ry 0 rz -180 deg; joints [0, 0, 0, 0, 0, 0]
  Call Extruder 0.02048
  MoveL (T199) to (103.79, 119.28, 0.3) mm, rotated rx 180 ry 0 rz -180 deg; joints [0, 0, 0, 0, 0, 0]
  Call Extruder 0.11008
  MoveL (T200) to (105.72, 121.21, 0.3) mm, rotated rx 180 ry 0 rz -180 deg; joints [0, 0, 0, 0, 0, 0]
  Call Extruder 0.02048
  MoveL (T201) to (105.21, 121.21, 0.3) mm, rotated rx 180 ry 0 rz -180 deg; joints [0, 0, 0, 0, 0, 0]
  Call Extruder 0.08111
  MoveL (T202) to (103.79, 119.79, 0.3) mm, rotated rx 180 ry 0 rz -180 deg; joints [0, 0, 0, 0, 0, 0]
  Call Extruder 0.02048
  MoveL (T203) to (103.79, 120.3, 0.3) mm, rotated rx 180 ry 0 rz -180 deg; joints [0, 0, 0, 0, 0, 0]
  Call Extruder 0.05214
  MoveL (T204) to (104.7, 121.21, 0.3) mm, rotated rx 180 ry 0 rz -180 deg; joints [0, 0, 0, 0, 0, 0]
  Call Extruder 0.02048
  MoveL (T205) to (104.19, 121.21, 0.3) mm, rotated rx 180 ry 0 rz -180 deg; joints [0, 0, 0, 0, 0, 0]
  Call Extruder 0.0323
  MoveL (T206) to (103.63, 120.65, 0.3) mm, rotated rx 180 ry 0 rz -180 deg; joints [0, 0, 0, 0, 0, 0]
  Set speed (45.0 mm/s)
  Call Extruder -1.6
  MoveL (T207) to (103.63, 120.65, 0.3) mm, rotated rx 180 ry 0 rz -180 deg; joints [0, 0, 0, 0, 0, 0]
  Set speed (120.0 mm/s)
  MoveL (T208) to (103.63, 120.65, 0.3) mm, rotated rx 180 ry 0 rz -180 deg; joints [0, 0, 0, 0, 0, 0]
  Call Extruder -0.28537
  MoveL (T209) to (104.19, 121.21, 0.3) mm, rotated rx 180 ry 0 rz -180 deg; joints [0, 0, 0, 0, 0, 0]
  Call Extruder -0.09463
  MoveL (T210) to (104.46, 121.21, 0.3) mm, rotated rx 180 ry 0 rz -180 deg; joints [0, 0, 0, 0, 0, 0]
  Set speed (45.0 mm/s)
  Call Extruder -0.02
  MoveL (T211) to (104.46, 121.21, 0.3) mm, rotated rx 180 ry 0 rz -180 deg; joints [0, 0, 0, 0, 0, 0]
  Set speed (150.0 mm/s)
  MoveL (T212) to (104.46, 121.21, 2.3) mm, rotated rx 180 ry 0 rz -180 deg; joints [0, 0, 0, 0, 0, 0]
  Call Mcode M104 S205
  MoveL (T213) to (104.46, 121.21, 2.3) mm, rotated rx 180 ry 0 rz -180 deg; joints [0, 0, 0, 0, 0, 0]
  Call Mcode M140 S60
  MoveL (T214) to (104.46, 121.21, 2.3) mm, rotated rx 180 ry 0 rz -180 deg; joints [0, 0, 0, 0, 0, 0]
  MoveL (T215) to (104.46, 125.86, 2.3) mm, rotated rx 180 ry 0 rz -180 deg; joints [0, 0, 0, 0, 0, 0]
  MoveL (T216) to (104.46, 125.86, 0.5) mm, rotated rx 180 ry 0 rz -180 deg; joints [0, 0, 0, 0, 0, 0]
  Set speed (40.0 mm/s)
  Call Extruder 2.0
  MoveL (T217) to (104.46, 125.86, 0.5) mm, rotated rx 180 ry 0 rz -180 deg; joints [0, 0, 0, 0, 0, 0]
  Set speed (25.0 mm/s)
  MoveL (T218) to (104.46, 125.86, 0.5) mm, rotated rx 180 ry 0 rz -180 deg; joints [0, 0, 0, 0, 0, 0]
  Call Extruder 0.05531
  MoveL (T219) to (102.5, 125.86, 0.5) mm, rotated rx 180 ry 0 rz -180 deg; joints [0, 0, 0, 0, 0, 0]
  Call Extruder 0.04589
  MoveL (T220) to (100.92, 125.46, 0.5) mm, rotated rx 180 ry 0 rz -180 deg; joints [0, 0, 0, 0, 0, 0]
  Call Extruder 0.04589
  MoveL (T221) to (99.72, 124.37, 0.5) mm, rotated rx 180 ry 0 rz -180 deg; joints [0, 0, 0, 0, 0, 0]
  Call Extruder 0.05523
  MoveL (T222) to (99.14, 122.5, 0.5) mm, rotated rx 180 ry 0 rz -180 deg; joints [0, 0, 0, 0, 0, 0]
  Call Extruder 0.56438
  MoveL (T223) to (99.14, 102.5, 0.5) mm, rotated rx 180 ry 0 rz -180 deg; joints [0, 0, 0, 0, 0, 0]
  Call Extruder 0.04589
  MoveL (T224) to (99.54, 100.92, 0.5) mm, rotated rx 180 ry 0 rz -180 deg; joints [0, 0, 0, 0, 0, 0]
  Call Extruder 0.04589
  MoveL (T225) to (100.63, 99.72, 0.5) mm, rotated rx 180 ry 0 rz -180 deg; joints [0, 0, 0, 0, 0, 0]
  Call Extruder 0.05523
  MoveL (T226) to (102.5, 99.14, 0.5) mm, rotated rx 180 ry 0 rz -180 deg; joints [0, 0, 0, 0, 0, 0]
  Call Extruder 0.56438
  MoveL (T227) to (122.5, 99.14, 0.5) mm, rotated rx 180 ry 0 rz -180 deg; joints [0, 0, 0, 0, 0, 0]
  Call Extruder 0.04589
  MoveL (T228) to (124.08, 99.54, 0.5) mm, rotated rx 180 ry 0 rz -180 deg; joints [0, 0, 0, 0, 0, 0]
  Call Extruder 0.04589
  MoveL (T229) to (125.28, 100.63, 0.5) mm, rotated rx 180 ry 0 rz -180 deg; joints [0, 0, 0, 0, 0, 0]
  Call Extruder 0.05523
  MoveL (T230) to (125.86, 102.5, 0.5) mm, rotated rx 180 ry 0 rz -180 deg; joints [0, 0, 0, 0, 0, 0]
  Call Extruder 0.56438
  MoveL (T231) to (125.86, 122.5, 0.5) mm, rotated rx 180 ry 0 rz -180 deg; joints [0, 0, 0, 0, 0, 0]
  Call Extruder 0.04589
  MoveL (T232) to (125.46, 124.08, 0.5) mm, rotated rx 180 ry 0 rz -180 deg; joints [0, 0, 0, 0, 0, 0]
  Call Extruder 0.04589
  MoveL (T233) to (124.37, 125.28, 0.5) mm, rotated rx 180 ry 0 rz -180 deg; joints [0, 0, 0, 0, 0, 0]
  Call Extruder 0.05523
  MoveL (T234) to (122.5, 125.86, 0.5) mm, rotated rx 180 ry 0 rz -180 deg; joints [0, 0, 0, 0, 0, 0]
  Call Extruder 0.50738
  MoveL (T235) to (104.52, 125.86, 0.5) mm, rotated rx 180 ry 0 rz -180 deg; joints [0, 0, 0, 0, 0, 0]
  Set speed (45.0 mm/s)
  Call Extruder -1.6
  MoveL (T236) to (104.52, 125.86, 0.5) mm, rotated rx 180 ry 0 rz -180 deg; joints [0, 0, 0, 0, 0, 0]
  Set speed (120.0 mm/s)
  MoveL (T237) to (104.52, 125.86, 0.5) mm, rotated rx 180 ry 0 rz -180 deg; joints [0, 0, 0, 0, 0, 0]
  Call Extruder -0.38
  MoveL (T238) to (103.45, 125.86, 0.5) mm, rotated rx 180 ry 0 rz -180 deg; joints [0, 0, 0, 0, 0, 0]
  Set speed (45.0 mm/s)
  Call Extruder -0.02
  MoveL (T239) to (103.45, 125.86, 0.5) mm, rotated rx 180 ry 0 rz -180 deg; joints [0, 0, 0, 0, 0, 0]
  Set speed (150.0 mm/s)
  MoveL (T240) to (103.45, 125.86, 2.5) mm, rotated rx 180 ry 0 rz -180 deg; joints [0, 0, 0, 0, 0, 0]
  MoveL (T241) to (104.34, 103.54, 2.5) mm, rotated rx 180 ry 0 rz -180 deg; joints [0, 0, 0, 0, 0, 0]
  MoveL (T242) to (104.34, 103.54, 0.5) mm, rotated rx 180 ry 0 rz -180 deg; joints [0, 0, 0, 0, 0, 0]
  Set speed (40.0 mm/s)
  Call Extruder 2.0
  MoveL (T243) to (104.34, 103.54, 0.5) mm, rotated rx 180 ry 0 rz -180 deg; joints [0, 0, 0, 0, 0, 0]
  Call Extruder 0.52159
  MoveL (T244) to (121.46, 103.54, 0.5) mm, rotated rx 180 ry 0 rz -180 deg; joints [0, 0, 0, 0, 0, 0]
  Call Extruder 0.54596
  MoveL (T245) to (121.46, 121.46, 0.5) mm, rotated rx 180 ry 0 rz -180 deg; joints [0, 0, 0, 0, 0, 0]
  Call Extruder 0.54596
  MoveL (T246) to (103.54, 121.46, 0.5) mm, rotated rx 180 ry 0 rz -180 deg; joints [0, 0, 0, 0, 0, 0]
  Call Extruder 0.54596
  MoveL (T247) to (103.54, 103.54, 0.5) mm, rotated rx 180 ry 0 rz -180 deg; joints [0, 0, 0, 0, 0, 0]
  Call Extruder 0.02254
  MoveL (T248) to (104.28, 103.54, 0.5) mm, rotated rx 180 ry 0 rz -180 deg; joints [0, 0, 0, 0, 0, 0]
  Set speed (150.0 mm/s)
  MoveL (T249) to (103.53, 103.13, 0.5) mm, rotated rx 180 ry 0 rz -180 deg; joints [0, 0, 0, 0, 0, 0]
  Set speed (40.0 mm/s)
  MoveL (T250) to (103.53, 103.13, 0.5) mm, rotated rx 180 ry 0 rz -180 deg; joints [0, 0, 0, 0, 0, 0]
  Call Extruder 0.55858
  MoveL (T251) to (121.87, 103.13, 0.5) mm, rotated rx 180 ry 0 rz -180 deg; joints [0, 0, 0, 0, 0, 0]
  Call Extruder 0.57077
  MoveL (T252) to (121.87, 121.87, 0.5) mm, rotated rx 180 ry 0 rz -180 deg; joints [0, 0, 0, 0, 0, 0]
  Call Extruder 0.57077
  MoveL (T253) to (103.13, 121.87, 0.5) mm, rotated rx 180 ry 0 rz -180 deg; joints [0, 0, 0, 0, 0, 0]
  Call Extruder 0.57077
  MoveL (T254) to (103.13, 103.13, 0.5) mm, rotated rx 180 ry 0 rz -180 deg; joints [0, 0, 0, 0, 0, 0]
  Call Extruder 0.01036
  MoveL (T255) to (103.47, 103.13, 0.5) mm, rotated rx 180 ry 0 rz -180 deg; joints [0, 0, 0, 0, 0, 0]
  Set speed (150.0 mm/s)
  MoveL (T256) to (102.72, 102.81, 0.5) mm, rotated rx 180 ry 0 rz -180 deg; joints [0, 0, 0, 0, 0, 0]
  Set speed (25.0 mm/s)
  MoveL (T257) to (102.72, 102.81, 0.5) mm, rotated rx 180 ry 0 rz -180 deg; joints [0, 0, 0, 0, 0, 0]
  Call Extruder 0.00259
  MoveL (T258) to (102.72, 102.72, 0.5) mm, rotated rx 180 ry 0 rz -180 deg; joints [0, 0, 0, 0, 0, 0]
  Call Extruder 0.59557
  MoveL (T259) to (122.28, 102.72, 0.5) mm, rotated rx 180 ry 0 rz -180 deg; joints [0, 0, 0, 0, 0, 0]
  Call Extruder 0.59557
  MoveL (T260) to (122.28, 122.28, 0.5) mm, rotated rx 180 ry 0 rz -180 deg; joints [0, 0, 0, 0, 0, 0]
  Call Extruder 0.59557
  MoveL (T261) to (102.72, 122.28, 0.5) mm, rotated rx 180 ry 0 rz -180 deg; joints [0, 0, 0, 0, 0, 0]
  Call Extruder 0.59115
  MoveL (T262) to (102.72, 102.87, 0.5) mm, rotated rx 180 ry 0 rz -180 deg; joints [0, 0, 0, 0, 0, 0]
  Set speed (150.0 mm/s)
  MoveL (T263) to (102.78, 102.75, 0.5) mm, rotated rx 180 ry 0 rz -180 deg; joints [0, 0, 0, 0, 0, 0]
  Set speed (45.0 mm/s)
  Call Extruder -1.6
  MoveL (T264) to (102.78, 102.75, 0.5) mm, rotated rx 180 ry 0 rz -180 deg; joints [0, 0, 0, 0, 0, 0]
  Set speed (120.0 mm/s)
  MoveL (T265) to (102.78, 102.75, 0.5) mm, rotated rx 180 ry 0 rz -180 deg; joints [0, 0, 0, 0, 0, 0]
  Call Extruder -0.05166
  MoveL (T266) to (102.72, 102.72, 0.5) mm, rotated rx 180 ry 0 rz -180 deg; joints [0, 0, 0, 0, 0, 0]
  Call Extruder -0.32834
  MoveL (T267) to (103.65, 102.72, 0.5) mm, rotated rx 180 ry 0 rz -180 deg; joints [0, 0, 0, 0, 0, 0]
  Set speed (45.0 mm/s)
  Call Extruder -0.02
  MoveL (T268) to (103.65, 102.72, 0.5) mm, rotated rx 180 ry 0 rz -180 deg; joints [0, 0, 0, 0, 0, 0]
  Set speed (150.0 mm/s)
  MoveL (T269) to (103.65, 102.72, 2.5) mm, rotated rx 180 ry 0 rz -180 deg; joints [0, 0, 0, 0, 0, 0]
  MoveL (T270) to (121.34, 120.51, 2.5) mm, rotated rx 180 ry 0 rz -180 deg; joints [0, 0, 0, 0, 0, 0]
  MoveL (T271) to (121.34, 120.51, 0.5) mm, rotated rx 180 ry 0 rz -180 deg; joints [0, 0, 0, 0, 0, 0]
  Set speed (40.0 mm/s)
  Call Extruder 2.0
  MoveL (T272) to (121.34, 120.51, 0.5) mm, rotated rx 180 ry 0 rz -180 deg; joints [0, 0, 0, 0, 0, 0]
  Call Extruder 0.02815
  MoveL (T273) to (120.69, 121.16, 0.5) mm, rotated rx 180 ry 0 rz -180 deg; joints [0, 0, 0, 0, 0, 0]
  Call Extruder 0.01786
  MoveL (T274) to (120.11, 121.16, 0.5) mm, rotated rx 180 ry 0 rz -180 deg; joints [0, 0, 0, 0, 0, 0]
  Call Extruder 0.04544
  MoveL (T275) to (121.16, 120.11, 0.5) mm, rotated rx 180 ry 0 rz -180 deg; joints [0, 0, 0, 0, 0, 0]
  Call Extruder 0.01786
  MoveL (T276) to (121.16, 119.53, 0.5) mm, rotated rx 180 ry 0 rz -180 deg; joints [0, 0, 0, 0, 0, 0]
  Call Extruder 0.0707
  MoveL (T277) to (119.53, 121.16, 0.5) mm, rotated rx 180 ry 0 rz -180 deg; joints [0, 0, 0, 0, 0, 0]
  Call Extruder 0.01786
  MoveL (T278) to (118.95, 121.16, 0.5) mm, rotated rx 180 ry 0 rz -180 deg; joints [0, 0, 0, 0, 0, 0]
  Call Extruder 0.09595
  MoveL (T279) to (121.16, 118.95, 0.5) mm, rotated rx 180 ry 0 rz -180 deg; joints [0, 0, 0, 0, 0, 0]
  Call Extruder 0.01786
  MoveL (T280) to (121.16, 118.37, 0.5) mm, rotated rx 180 ry 0 rz -180 deg; joints [0, 0, 0, 0, 0, 0]
  Call Extruder 0.12121
  MoveL (T281) to (118.37, 121.16, 0.5) mm, rotated rx 180 ry 0 rz -180 deg; joints [0, 0, 0, 0, 0, 0]
  Call Extruder 0.01786
  MoveL (T282) to (117.79, 121.16, 0.5) mm, rotated rx 180 ry 0 rz -180 deg; joints [0, 0, 0, 0, 0, 0]
  Call Extruder 0.14646
  MoveL (T283) to (121.16, 117.79, 0.5) mm, rotated rx 180 ry 0 rz -180 deg; joints [0, 0, 0, 0, 0, 0]
  Call Extruder 0.01786
  MoveL (T284) to (121.16, 117.21, 0.5) mm, rotated rx 180 ry 0 rz -180 deg; joints [0, 0, 0, 0, 0, 0]
  Call Extruder 0.17172
  MoveL (T285) to (117.21, 121.16, 0.5) mm, rotated rx 180 ry 0 rz -180 deg; joints [0, 0, 0, 0, 0, 0]
  Call Extruder 0.01786
  MoveL (T286) to (116.62, 121.16, 0.5) mm, rotated rx 180 ry 0 rz -180 deg; joints [0, 0, 0, 0, 0, 0]
  Call Extruder 0.19697
  MoveL (T287) to (121.16, 116.62, 0.5) mm, rotated rx 180 ry 0 rz -180 deg; joints [0, 0, 0, 0, 0, 0]
  Call Extruder 0.01786
  MoveL (T288) to (121.16, 116.04, 0.5) mm, rotated rx 180 ry 0 rz -180 deg; joints [0, 0, 0, 0, 0, 0]
  Call Extruder 0.22223
  MoveL (T289) to (116.04, 121.16, 0.5) mm, rotated rx 180 ry 0 rz -180 deg; joints [0, 0, 0, 0, 0, 0]
  Call Extruder 0.01786
  MoveL (T290) to (115.46, 121.16, 0.5) mm, rotated rx 180 ry 0 rz -180 deg; joints [0, 0, 0, 0, 0, 0]
  Call Extruder 0.24748
  MoveL (T291) to (121.16, 115.46, 0.5) mm, rotated rx 180 ry 0 rz -180 deg; joints [0, 0, 0, 0, 0, 0]
  Call Extruder 0.01786
  MoveL (T292) to (121.16, 114.88, 0.5) mm, rotated rx 180 ry 0 rz -180 deg; joints [0, 0, 0, 0, 0, 0]
  Call Extruder 0.27274
  MoveL (T293) to (114.88, 121.16, 0.5) mm, rotated rx 180 ry 0 rz -180 deg; joints [0, 0, 0, 0, 0, 0]
  Call Extruder 0.01786
  MoveL (T294) to (114.3, 121.16, 0.5) mm, rotated rx 180 ry 0 rz -180 deg; joints [0, 0, 0, 0, 0, 0]
  Call Extruder 0.29799
  MoveL (T295) to (121.16, 114.3, 0.5) mm, rotated rx 180 ry 0 rz -180 deg; joints [0, 0, 0, 0, 0, 0]
  Call Extruder 0.01786
  MoveL (T296) to (121.16, 113.72, 0.5) mm, rotated rx 180 ry 0 rz -180 deg; joints [0, 0, 0, 0, 0, 0]
  Call Extruder 0.32324
  MoveL (T297) to (113.72, 121.16, 0.5) mm, rotated rx 180 ry 0 rz -180 deg; joints [0, 0, 0, 0, 0, 0]
  Call Extruder 0.01786
  MoveL (T298) to (113.14, 121.16, 0.5) mm, rotated rx 180 ry 0 rz -180 deg; joints [0, 0, 0, 0, 0, 0]
  Call Extruder 0.3485
  MoveL (T299) to (121.16, 113.14, 0.5) mm, rotated rx 180 ry 0 rz -180 deg; joints [0, 0, 0, 0, 0, 0]
  Call Extruder 0.01786
  MoveL (T300) to (121.16, 112.56, 0.5) mm, rotated rx 180 ry 0 rz -180 deg; joints [0, 0, 0, 0, 0, 0]
  Call Extruder 0.37375
  MoveL (T301) to (112.56, 121.16, 0.5) mm, rotated rx 180 ry 0 rz -180 deg; joints [0, 0, 0, 0, 0, 0]
  Call Extruder 0.01786
  MoveL (T302) to (111.98, 121.16, 0.5) mm, rotated rx 180 ry 0 rz -180 deg; joints [0, 0, 0, 0, 0, 0]
  Call Extruder 0.39901
  MoveL (T303) to (121.16, 111.98, 0.5) mm, rotated rx 180 ry 0 rz -180 deg; joints [0, 0, 0, 0, 0, 0]
  Call Extruder 0.01786
  MoveL (T304) to (121.16, 111.4, 0.5) mm, rotated rx 180 ry 0 rz -180 deg; joints [0, 0, 0, 0, 0, 0]
  Call Extruder 0.42426
  MoveL (T305) to (111.4, 121.16, 0.5) mm, rotated rx 180 ry 0 rz -180 deg; joints [0, 0, 0, 0, 0, 0]
  Call Extruder 0.01786
  MoveL (T306) to (110.81, 121.16, 0.5) mm, rotated rx 180 ry 0 rz -180 deg; joints [0, 0, 0, 0, 0, 0]
  Call Extruder 0.44952
  MoveL (T307) to (121.16, 110.81, 0.5) mm, rotated rx 180 ry 0 rz -180 deg; joints [0, 0, 0, 0, 0, 0]
  Call Extruder 0.01786
  MoveL (T308) to (121.16, 110.23, 0.5) mm, rotated rx 180 ry 0 rz -180 deg; joints [0, 0, 0, 0, 0, 0]
  Call Extruder 0.47477
  MoveL (T309) to (110.23, 121.16, 0.5) mm, rotated rx 180 ry 0 rz -180 deg; joints [0, 0, 0, 0, 0, 0]
  Call Extruder 0.01786
  MoveL (T310) to (109.65, 121.16, 0.5) mm, rotated rx 180 ry 0 rz -180 deg; joints [0, 0, 0, 0, 0, 0]
  Call Extruder 0.50003
  MoveL (T311) to (121.16, 109.65, 0.5) mm, rotated rx 180 ry 0 rz -180 deg; joints [0, 0, 0, 0, 0, 0]
  Call Extruder 0.01786
  MoveL (T312) to (121.16, 109.07, 0.5) mm, rotated rx 180 ry 0 rz -180 deg; joints [0, 0, 0, 0, 0, 0]
  Call Extruder 0.52528
  MoveL (T313) to (109.07, 121.16, 0.5) mm, rotated rx 180 ry 0 rz -180 deg; joints [0, 0, 0, 0, 0, 0]
  Call Extruder 0.01786
  MoveL (T314) to (108.49, 121.16, 0.5) mm, rotated rx 180 ry 0 rz -180 deg; joints [0, 0, 0, 0, 0, 0]
  Call Extruder 0.55054
  MoveL (T315) to (121.16, 108.49, 0.5) mm, rotated rx 180 ry 0 rz -180 deg; joints [0, 0, 0, 0, 0, 0]
  Call Extruder 0.01786
  MoveL (T316) to (121.16, 107.91, 0.5) mm, rotated rx 180 ry 0 rz -180 deg; joints [0, 0, 0, 0, 0, 0]
  Call Extruder 0.57579
  MoveL (T317) to (107.91, 121.16, 0.5) mm, rotated rx 180 ry 0 rz -180 deg; joints [0, 0, 0, 0, 0, 0]
  Call Extruder 0.01786
  MoveL (T318) to (107.33, 121.16, 0.5) mm, rotated rx 180 ry 0 rz -180 deg; joints [0, 0, 0, 0, 0, 0]
  Call Extruder 0.60105
  MoveL (T319) to (121.16, 107.33, 0.5) mm, rotated rx 180 ry 0 rz -180 deg; joints [0, 0, 0, 0, 0, 0]
  Call Extruder 0.01786
  MoveL (T320) to (121.16, 106.75, 0.5) mm, rotated rx 180 ry 0 rz -180 deg; joints [0, 0, 0, 0, 0, 0]
  Call Extruder 0.6263
  MoveL (T321) to (106.75, 121.16, 0.5) mm, rotated rx 180 ry 0 rz -180 deg; joints [0, 0, 0, 0, 0, 0]
  Call Extruder 0.01786
  MoveL (T322) to (106.17, 121.16, 0.5) mm, rotated rx 180 ry 0 rz -180 deg; joints [0, 0, 0, 0, 0, 0]
  Call Extruder 0.65156
  MoveL (T323) to (121.16, 106.17, 0.5) mm, rotated rx 180 ry 0 rz -180 deg; joints [0, 0, 0, 0, 0, 0]
  Call Extruder 0.01786
  MoveL (T324) to (121.16, 105.59, 0.5) mm, rotated rx 180 ry 0 rz -180 deg; joints [0, 0, 0, 0, 0, 0]
  Call Extruder 0.67681
  MoveL (T325) to (105.59, 121.16, 0.5) mm, rotated rx 180 ry 0 rz -180 deg; joints [0, 0, 0, 0, 0, 0]
  Call Extruder 0.01786
  MoveL (T326) to (105.01, 121.16, 0.5) mm, rotated rx 180 ry 0 rz -180 deg; joints [0, 0, 0, 0, 0, 0]
  Call Extruder 0.70207
  MoveL (T327) to (121.16, 105.01, 0.5) mm, rotated rx 180 ry 0 rz -180 deg; joints [0, 0, 0, 0, 0, 0]
  Call Extruder 0.01786
  MoveL (T328) to (121.16, 104.42, 0.5) mm, rotated rx 180 ry 0 rz -180 deg; joints [0, 0, 0, 0, 0, 0]
  Call Extruder 0.72732
  MoveL (T329) to (104.42, 121.16, 0.5) mm, rotated rx 180 ry 0 rz -180 deg; joints [0, 0, 0, 0, 0, 0]
  Call Extruder 0.01786
  MoveL (T330) to (103.84, 121.16, 0.5) mm, rotated rx 180 ry 0 rz -180 deg; joints [0, 0, 0, 0, 0, 0]
  Call Extruder 0.75257
  MoveL (T331) to (121.16, 103.84, 0.5) mm, rotated rx 180 ry 0 rz -180 deg; joints [0, 0, 0, 0, 0, 0]
  Call Extruder 0.01786
  MoveL (T332) to (120.58, 103.84, 0.5) mm, rotated rx 180 ry 0 rz -180 deg; joints [0, 0, 0, 0, 0, 0]
  Call Extruder 0.72732
  MoveL (T333) to (103.84, 120.58, 0.5) mm, rotated rx 180 ry 0 rz -180 deg; joints [0, 0, 0, 0, 0, 0]
  Call Extruder 0.01786
  MoveL (T334) to (103.84, 119.99, 0.5) mm, rotated rx 180 ry 0 rz -180 deg; joints [0, 0, 0, 0, 0, 0]
  Call Extruder 0.70206
  MoveL (T335) to (119.99, 103.84, 0.5) mm, rotated rx 180 ry 0 rz -180 deg; joints [0, 0, 0, 0, 0, 0]
  Call Extruder 0.01786
  MoveL (T336) to (119.41, 103.84, 0.5) mm, rotated rx 180 ry 0 rz -180 deg; joints [0, 0, 0, 0, 0, 0]
  Call Extruder 0.67681
  MoveL (T337) to (103.84, 119.41, 0.5) mm, rotated rx 180 ry 0 rz -180 deg; joints [0, 0, 0, 0, 0, 0]
  Call Extruder 0.01786
  MoveL (T338) to (103.84, 118.83, 0.5) mm, rotated rx 180 ry 0 rz -180 deg; joints [0, 0, 0, 0, 0, 0]
  Call Extruder 0.65155
  MoveL (T339) to (118.83, 103.84, 0.5) mm, rotated rx 180 ry 0 rz -180 deg; joints [0, 0, 0, 0, 0, 0]
  Call Extruder 0.01786
  MoveL (T340) to (118.25, 103.84, 0.5) mm, rotated rx 180 ry 0 rz -180 deg; joints [0, 0, 0, 0, 0, 0]
  Call Extruder 0.6263
  MoveL (T341) to (103.84, 118.25, 0.5) mm, rotated rx 180 ry 0 rz -180 deg; joints [0, 0, 0, 0, 0, 0]
  Call Extruder 0.01786
  MoveL (T342) to (103.84, 117.67, 0.5) mm, rotated rx 180 ry 0 rz -180 deg; joints [0, 0, 0, 0, 0, 0]
  Call Extruder 0.60104
  MoveL (T343) to (117.67, 103.84, 0.5) mm, rotated rx 180 ry 0 rz -180 deg; joints [0, 0, 0, 0, 0, 0]
  Call Extruder 0.01786
  MoveL (T344) to (117.09, 103.84, 0.5) mm, rotated rx 180 ry 0 rz -180 deg; joints [0, 0, 0, 0, 0, 0]
  Call Extruder 0.57579
  MoveL (T345) to (103.84, 117.09, 0.5) mm, rotated rx 180 ry 0 rz -180 deg; joints [0, 0, 0, 0, 0, 0]
  Call Extruder 0.01786
  MoveL (T346) to (103.84, 116.51, 0.5) mm, rotated rx 180 ry 0 rz -180 deg; joints [0, 0, 0, 0, 0, 0]
  Call Extruder 0.55053
  MoveL (T347) to (116.51, 103.84, 0.5) mm, rotated rx 180 ry 0 rz -180 deg; joints [0, 0, 0, 0, 0, 0]
  Call Extruder 0.01786
  MoveL (T348) to (115.93, 103.84, 0.5) mm, rotated rx 180 ry 0 rz -180 deg; joints [0, 0, 0, 0, 0, 0]
  Call Extruder 0.52528
  MoveL (T349) to (103.84, 115.93, 0.5) mm, rotated rx 180 ry 0 rz -180 deg; joints [0, 0, 0, 0, 0, 0]
  Call Extruder 0.01786
  MoveL (T350) to (103.84, 115.35, 0.5) mm, rotated rx 180 ry 0 rz -180 deg; joints [0, 0, 0, 0, 0, 0]
  Call Extruder 0.50002
  MoveL (T351) to (115.35, 103.84, 0.5) mm, rotated rx 180 ry 0 rz -180 deg; joints [0, 0, 0, 0, 0, 0]
  Call Extruder 0.01786
  MoveL (T352) to (114.77, 103.84, 0.5) mm, rotated rx 180 ry 0 rz -180 deg; joints [0, 0, 0, 0, 0, 0]
  Call Extruder 0.47477
  MoveL (T353) to (103.84, 114.77, 0.5) mm, rotated rx 180 ry 0 rz -180 deg; joints [0, 0, 0, 0, 0, 0]
  Call Extruder 0.01786
  MoveL (T354) to (103.84, 114.18, 0.5) mm, rotated rx 180 ry 0 rz -180 deg; joints [0, 0, 0, 0, 0, 0]
  Call Extruder 0.44951
  MoveL (T355) to (114.18, 103.84, 0.5) mm, rotated rx 180 ry 0 rz -180 deg; joints [0, 0, 0, 0, 0, 0]
  Call Extruder 0.01786
  MoveL (T356) to (113.6, 103.84, 0.5) mm, rotated rx 180 ry 0 rz -180 deg; joints [0, 0, 0, 0, 0, 0]
  Call Extruder 0.42426
  MoveL (T357) to (103.84, 113.6, 0.5) mm, rotated rx 180 ry 0 rz -180 deg; joints [0, 0, 0, 0, 0, 0]
  Call Extruder 0.01786
  MoveL (T358) to (103.84, 113.02, 0.5) mm, rotated rx 180 ry 0 rz -180 deg; joints [0, 0, 0, 0, 0, 0]
  Call Extruder 0.399
  MoveL (T359) to (113.02, 103.84, 0.5) mm, rotated rx 180 ry 0 rz -180 deg; joints [0, 0, 0, 0, 0, 0]
  Call Extruder 0.01786
  MoveL (T360) to (112.44, 103.84, 0.5) mm, rotated rx 180 ry 0 rz -180 deg; joints [0, 0, 0, 0, 0, 0]
  Call Extruder 0.37375
  MoveL (T361) to (103.84, 112.44, 0.5) mm, rotated rx 180 ry 0 rz -180 deg; joints [0, 0, 0, 0, 0, 0]
  Call Extruder 0.01786
  MoveL (T362) to (103.84, 111.86, 0.5) mm, rotated rx 180 ry 0 rz -180 deg; joints [0, 0, 0, 0, 0, 0]
  Call Extruder 0.3485
  MoveL (T363) to (111.86, 103.84, 0.5) mm, rotated rx 180 ry 0 rz -180 deg; joints [0, 0, 0, 0, 0, 0]
  Call Extruder 0.01786
  MoveL (T364) to (111.28, 103.84, 0.5) mm, rotated rx 180 ry 0 rz -180 deg; joints [0, 0, 0, 0, 0, 0]
  Call Extruder 0.32324
  MoveL (T365) to (103.84, 111.28, 0.5) mm, rotated rx 180 ry 0 rz -180 deg; joints [0, 0, 0, 0, 0, 0]
  Call Extruder 0.01786
  MoveL (T366) to (103.84, 110.7, 0.5) mm, rotated rx 180 ry 0 rz -180 deg; joints [0, 0, 0, 0, 0, 0]
  Call Extruder 0.29799
  MoveL (T367) to (110.7, 103.84, 0.5) mm, rotated rx 180 ry 0 rz -180 deg; joints [0, 0, 0, 0, 0, 0]
  Call Extruder 0.01786
  MoveL (T368) to (110.12, 103.84, 0.5) mm, rotated rx 180 ry 0 rz -180 deg; joints [0, 0, 0, 0, 0, 0]
  Call Extruder 0.27273
  MoveL (T369) to (103.84, 110.12, 0.5) mm, rotated rx 180 ry 0 rz -180 deg; joints [0, 0, 0, 0, 0, 0]
  Call Extruder 0.01786
  MoveL (T370) to (103.84, 109.54, 0.5) mm, rotated rx 180 ry 0 rz -180 deg; joints [0, 0, 0, 0, 0, 0]
  Call Extruder 0.24748
  MoveL (T371) to (109.54, 103.84, 0.5) mm, rotated rx 180 ry 0 rz -180 deg; joints [0, 0, 0, 0, 0, 0]
  Call Extruder 0.01786
  MoveL (T372) to (108.96, 103.84, 0.5) mm, rotated rx 180 ry 0 rz -180 deg; joints [0, 0, 0, 0, 0, 0]
  Call Extruder 0.22222
  MoveL (T373) to (103.84, 108.96, 0.5) mm, rotated rx 180 ry 0 rz -180 deg; joints [0, 0, 0, 0, 0, 0]
  Call Extruder 0.01786
  MoveL (T374) to (103.84, 108.38, 0.5) mm, rotated rx 180 ry 0 rz -180 deg; joints [0, 0, 0, 0, 0, 0]
  Call Extruder 0.19697
  MoveL (T375) to (108.38, 103.84, 0.5) mm, rotated rx 180 ry 0 rz -180 deg; joints [0, 0, 0, 0, 0, 0]
  Call Extruder 0.01786
  MoveL (T376) to (107.79, 103.84, 0.5) mm, rotated rx 180 ry 0 rz -180 deg; joints [0, 0, 0, 0, 0, 0]
  Call Extruder 0.17171
  MoveL (T377) to (103.84, 107.79, 0.5) mm, rotated rx 180 ry 0 rz -180 deg; joints [0, 0, 0, 0, 0, 0]
  Call Extruder 0.01786
  MoveL (T378) to (103.84, 107.21, 0.5) mm, rotated rx 180 ry 0 rz -180 deg; joints [0, 0, 0, 0, 0, 0]
  Call Extruder 0.14646
  MoveL (T379) to (107.21, 103.84, 0.5) mm, rotated rx 180 ry 0 rz -180 deg; joints [0, 0, 0, 0, 0, 0]
  Call Extruder 0.01786
  MoveL (T380) to (106.63, 103.84, 0.5) mm, rotated rx 180 ry 0 rz -180 deg; joints [0, 0, 0, 0, 0, 0]
  Call Extruder 0.1212
  MoveL (T381) to (103.84, 106.63, 0.5) mm, rotated rx 180 ry 0 rz -180 deg; joints [0, 0, 0, 0, 0, 0]
  Call Extruder 0.01786
  MoveL (T382) to (103.84, 106.05, 0.5) mm, rotated rx 180 ry 0 rz -180 deg; joints [0, 0, 0, 0, 0, 0]
  Call Extruder 0.09595
  MoveL (T383) to (106.05, 103.84, 0.5) mm, rotated rx 180 ry 0 rz -180 deg; joints [0, 0, 0, 0, 0, 0]
  Call Extruder 0.01786
  MoveL (T384) to (105.47, 103.84, 0.5) mm, rotated rx 180 ry 0 rz -180 deg; joints [0, 0, 0, 0, 0, 0]
  Call Extruder 0.07069
  MoveL (T385) to (103.84, 105.47, 0.5) mm, rotated rx 180 ry 0 rz -180 deg; joints [0, 0, 0, 0, 0, 0]
  Call Extruder 0.01786
  MoveL (T386) to (103.84, 104.89, 0.5) mm, rotated rx 180 ry 0 rz -180 deg; joints [0, 0, 0, 0, 0, 0]
  Call Extruder 0.04544
  MoveL (T387) to (104.89, 103.84, 0.5) mm, rotated rx 180 ry 0 rz -180 deg; joints [0, 0, 0, 0, 0, 0]
  Call Extruder 0.01786
  MoveL (T388) to (104.31, 103.84, 0.5) mm, rotated rx 180 ry 0 rz -180 deg; joints [0, 0, 0, 0, 0, 0]
  Call Extruder 0.02815
  MoveL (T389) to (103.66, 104.49, 0.5) mm, rotated rx 180 ry 0 rz -180 deg; joints [0, 0, 0, 0, 0, 0]
  Set speed (45.0 mm/s)
  Call Extruder -1.6
  MoveL (T390) to (103.66, 104.49, 0.5) mm, rotated rx 180 ry 0 rz -180 deg; joints [0, 0, 0, 0, 0, 0]
  Set speed (120.0 mm/s)
  MoveL (T391) to (103.66, 104.49, 0.5) mm, rotated rx 180 ry 0 rz -180 deg; joints [0, 0, 0, 0, 0, 0]
  Call Extruder -0.3262
  MoveL (T392) to (104.31, 103.84, 0.5) mm, rotated rx 180 ry 0 rz -180 deg; joints [0, 0, 0, 0, 0, 0]
  Call Extruder -0.0538
  MoveL (T393) to (104.46, 103.84, 0.5) mm, rotated rx 180 ry 0 rz -180 deg; joints [0, 0, 0, 0, 0, 0]
  Set speed (45.0 mm/s)
  Call Extruder -0.02
  MoveL (T394) to (104.46, 103.84, 0.5) mm, rotated rx 180 ry 0 rz -180 deg; joints [0, 0, 0, 0, 0, 0]
  Set speed (150.0 mm/s)
  MoveL (T395) to (104.46, 103.84, 2.5) mm, rotated rx 180 ry 0 rz -180 deg; joints [0, 0, 0, 0, 0, 0]
  MoveL (T396) to (104.34, 103.54, 2.5) mm, rotated rx 180 ry 0 rz -180 deg; joints [0, 0, 0, 0, 0, 0]
  MoveL (T397) to (104.34, 103.54, 0.7) mm, rotated rx 180 ry 0 rz -180 deg; joints [0, 0, 0, 0, 0, 0]
  Set speed (40.0 mm/s)
  Call Extruder 2.0
  MoveL (T398) to (104.34, 103.54, 0.7) mm, rotated rx 180 ry 0 rz -180 deg; joints [0, 0, 0, 0, 0, 0]
  Call Extruder 0.52159
  MoveL (T399) to (121.46, 103.54, 0.7) mm, rotated rx 180 ry 0 rz -180 deg; joints [0, 0, 0, 0, 0, 0]
  Call Extruder 0.54596
  MoveL (T400) to (121.46, 121.46, 0.7) mm, rotated rx 180 ry 0 rz -180 deg; joints [0, 0, 0, 0, 0, 0]
  Call Extruder 0.54596
  MoveL (T401) to (103.54, 121.46, 0.7) mm, rotated rx 180 ry 0 rz -180 deg; joints [0, 0, 0, 0, 0, 0]
  Call Extruder 0.54596
  MoveL (T402) to (103.54, 103.54, 0.7) mm, rotated rx 180 ry 0 rz -180 deg; joints [0, 0, 0, 0, 0, 0]
  Call Extruder 0.02254
  MoveL (T403) to (104.28, 103.54, 0.7) mm, rotated rx 180 ry 0 rz -180 deg; joints [0, 0, 0, 0, 0, 0]
  Set speed (150.0 mm/s)
  MoveL (T404) to (103.53, 103.13, 0.7) mm, rotated rx 180 ry 0 rz -180 deg; joints [0, 0, 0, 0, 0, 0]
  Set speed (40.0 mm/s)
  MoveL (T405) to (103.53, 103.13, 0.7) mm, rotated rx 180 ry 0 rz -180 deg; joints [0, 0, 0, 0, 0, 0]
  Call Extruder 0.55858
  MoveL (T406) to (121.87, 103.13, 0.7) mm, rotated rx 180 ry 0 rz -180 deg; joints [0, 0, 0, 0, 0, 0]
  Call Extruder 0.57077
  MoveL (T407) to (121.87, 121.87, 0.7) mm, rotated rx 180 ry 0 rz -180 deg; joints [0, 0, 0, 0, 0, 0]
  Call Extruder 0.57077
  MoveL (T408) to (103.13, 121.87, 0.7) mm, rotated rx 180 ry 0 rz -180 deg; joints [0, 0, 0, 0, 0, 0]
  Call Extruder 0.57077
  MoveL (T409) to (103.13, 103.13, 0.7) mm, rotated rx 180 ry 0 rz -180 deg; joints [0, 0, 0, 0, 0, 0]
  Call Extruder 0.01036
  MoveL (T410) to (103.47, 103.13, 0.7) mm, rotated rx 180 ry 0 rz -180 deg; joints [0, 0, 0, 0, 0, 0]
  Set speed (150.0 mm/s)
  MoveL (T411) to (102.72, 102.81, 0.7) mm, rotated rx 180 ry 0 rz -180 deg; joints [0, 0, 0, 0, 0, 0]
  Set speed (25.0 mm/s)
  MoveL (T412) to (102.72, 102.81, 0.7) mm, rotated rx 180 ry 0 rz -180 deg; joints [0, 0, 0, 0, 0, 0]
  Call Extruder 0.00259
  MoveL (T413) to (102.72, 102.72, 0.7) mm, rotated rx 180 ry 0 rz -180 deg; joints [0, 0, 0, 0, 0, 0]
  Call Extruder 0.59557
  MoveL (T414) to (122.28, 102.72, 0.7) mm, rotated rx 180 ry 0 rz -180 deg; joints [0, 0, 0, 0, 0, 0]
  Call Extruder 0.59557
  MoveL (T415) to (122.28, 122.28, 0.7) mm, rotated rx 180 ry 0 rz -180 deg; joints [0, 0, 0, 0, 0, 0]
  Call Extruder 0.59557
  MoveL (T416) to (102.72, 122.28, 0.7) mm, rotated rx 180 ry 0 rz -180 deg; joints [0, 0, 0, 0, 0, 0]
  Call Extruder 0.59115
  MoveL (T417) to (102.72, 102.87, 0.7) mm, rotated rx 180 ry 0 rz -180 deg; joints [0, 0, 0, 0, 0, 0]
  Set speed (150.0 mm/s)
  MoveL (T418) to (102.78, 102.75, 0.7) mm, rotated rx 180 ry 0 rz -180 deg; joints [0, 0, 0, 0, 0, 0]
  Set speed (45.0 mm/s)
  Call Extruder -1.6
  MoveL (T419) to (102.78, 102.75, 0.7) mm, rotated rx 180 ry 0 rz -180 deg; joints [0, 0, 0, 0, 0, 0]
  Set speed (120.0 mm/s)
  MoveL (T420) to (102.78, 102.75, 0.7) mm, rotated rx 180 ry 0 rz -180 deg; joints [0, 0, 0, 0, 0, 0]
  Call Extruder -0.05166
  MoveL (T421) to (102.72, 102.72, 0.7) mm, rotated rx 180 ry 0 rz -180 deg; joints [0, 0, 0, 0, 0, 0]
  Call Extruder -0.32834
  MoveL (T422) to (103.65, 102.72, 0.7) mm, rotated rx 180 ry 0 rz -180 deg; joints [0, 0, 0, 0, 0, 0]
  Set speed (45.0 mm/s)
  Call Extruder -0.02
  MoveL (T423) to (103.65, 102.72, 0.7) mm, rotated rx 180 ry 0 rz -180 deg; joints [0, 0, 0, 0, 0, 0]
  Set speed (150.0 mm/s)
  MoveL (T424) to (103.65, 102.72, 2.7) mm, rotated rx 180 ry 0 rz -180 deg; joints [0, 0, 0, 0, 0, 0]
  MoveL (T425) to (120.51, 103.66, 2.7) mm, rotated rx 180 ry 0 rz -180 deg; joints [0, 0, 0, 0, 0, 0]
  MoveL (T426) to (120.51, 103.66, 0.7) mm, rotated rx 180 ry 0 rz -180 deg; joints [0, 0, 0, 0, 0, 0]
  Set speed (40.0 mm/s)
  Call Extruder 2.0
  MoveL (T427) to (120.51, 103.66, 0.7) mm, rotated rx 180 ry 0 rz -180 deg; joints [0, 0, 0, 0, 0, 0]
  Call Extruder 0.02815
  MoveL (T428) to (121.16, 104.31, 0.7) mm, rotated rx 180 ry 0 rz -180 deg; joints [0, 0, 0, 0, 0, 0]
  Call Extruder 0.01786
  MoveL (T429) to (121.16, 104.89, 0.7) mm, rotated rx 180 ry 0 rz -180 deg; joints [0, 0, 0, 0, 0, 0]
  Call Extruder 0.04544
  MoveL (T430) to (120.11, 103.84, 0.7) mm, rotated rx 180 ry 0 rz -180 deg; joints [0, 0, 0, 0, 0, 0]
  Call Extruder 0.01786
  MoveL (T431) to (119.53, 103.84, 0.7) mm, rotated rx 180 ry 0 rz -180 deg; joints [0, 0, 0, 0, 0, 0]
  Call Extruder 0.0707
  MoveL (T432) to (121.16, 105.47, 0.7) mm, rotated rx 180 ry 0 rz -180 deg; joints [0, 0, 0, 0, 0, 0]
  Call Extruder 0.01786
  MoveL (T433) to (121.16, 106.05, 0.7) mm, rotated rx 180 ry 0 rz -180 deg; joints [0, 0, 0, 0, 0, 0]
  Call Extruder 0.09595
  MoveL (T434) to (118.95, 103.84, 0.7) mm, rotated rx 180 ry 0 rz -180 deg; joints [0, 0, 0, 0, 0, 0]
  Call Extruder 0.01786
  MoveL (T435) to (118.37, 103.84, 0.7) mm, rotated rx 180 ry 0 rz -180 deg; joints [0, 0, 0, 0, 0, 0]
  Call Extruder 0.12121
  MoveL (T436) to (121.16, 106.63, 0.7) mm, rotated rx 180 ry 0 rz -180 deg; joints [0, 0, 0, 0, 0, 0]
  Call Extruder 0.01786
  MoveL (T437) to (121.16, 107.21, 0.7) mm, rotated rx 180 ry 0 rz -180 deg; joints [0, 0, 0, 0, 0, 0]
  Call Extruder 0.14646
  MoveL (T438) to (117.79, 103.84, 0.7) mm, rotated rx 180 ry 0 rz -180 deg; joints [0, 0, 0, 0, 0, 0]
  Call Extruder 0.01786
  MoveL (T439) to (117.21, 103.84, 0.7) mm, rotated rx 180 ry 0 rz -180 deg; joints [0, 0, 0, 0, 0, 0]
  Call Extruder 0.17172
  MoveL (T440) to (121.16, 107.79, 0.7) mm, rotated rx 180 ry 0 rz -180 deg; joints [0, 0, 0, 0, 0, 0]
  Call Extruder 0.01786
  MoveL (T441) to (121.16, 108.38, 0.7) mm, rotated rx 180 ry 0 rz -180 deg; joints [0, 0, 0, 0, 0, 0]
  Call Extruder 0.19697
  MoveL (T442) to (116.62, 103.84, 0.7) mm, rotated rx 180 ry 0 rz -180 deg; joints [0, 0, 0, 0, 0, 0]
  Call Extruder 0.01786
  MoveL (T443) to (116.04, 103.84, 0.7) mm, rotated rx 180 ry 0 rz -180 deg; joints [0, 0, 0, 0, 0, 0]
  Call Extruder 0.22223
  MoveL (T444) to (121.16, 108.96, 0.7) mm, rotated rx 180 ry 0 rz -180 deg; joints [0, 0, 0, 0, 0, 0]
  Call Extruder 0.01786
  MoveL (T445) to (121.16, 109.54, 0.7) mm, rotated rx 180 ry 0 rz -180 deg; joints [0, 0, 0, 0, 0, 0]
  Call Extruder 0.24748
  MoveL (T446) to (115.46, 103.84, 0.7) mm, rotated rx 180 ry 0 rz -180 deg; joints [0, 0, 0, 0, 0, 0]
  Call Extruder 0.01786
  MoveL (T447) to (114.88, 103.84, 0.7) mm, rotated rx 180 ry 0 rz -180 deg; joints [0, 0, 0, 0, 0, 0]
  Call Extruder 0.27274
  MoveL (T448) to (121.16, 110.12, 0.7) mm, rotated rx 180 ry 0 rz -180 deg; joints [0, 0, 0, 0, 0, 0]
  Call Extruder 0.01786
  MoveL (T449) to (121.16, 110.7, 0.7) mm, rotated rx 180 ry 0 rz -180 deg; joints [0, 0, 0, 0, 0, 0]
  Call Extruder 0.29799
  MoveL (T450) to (114.3, 103.84, 0.7) mm, rotated rx 180 ry 0 rz -180 deg; joints [0, 0, 0, 0, 0, 0]
  Call Extruder 0.01786
  MoveL (T451) to (113.72, 103.84, 0.7) mm, rotated rx 180 ry 0 rz -180 deg; joints [0, 0, 0, 0, 0, 0]
  Call Extruder 0.32324
  MoveL (T452) to (121.16, 111.28, 0.7) mm, rotated rx 180 ry 0 rz -180 deg; joints [0, 0, 0, 0, 0, 0]
  Call Extruder 0.01786
  MoveL (T453) to (121.16, 111.86, 0.7) mm, rotated rx 180 ry 0 rz -180 deg; joints [0, 0, 0, 0, 0, 0]
  Call Extruder 0.3485
  MoveL (T454) to (113.14, 103.84, 0.7) mm, rotated rx 180 ry 0 rz -180 deg; joints [0, 0, 0, 0, 0, 0]
  Call Extruder 0.01786
  MoveL (T455) to (112.56, 103.84, 0.7) mm, rotated rx 180 ry 0 rz -180 deg; joints [0, 0, 0, 0, 0, 0]
  Call Extruder 0.37375
  MoveL (T456) to (121.16, 112.44, 0.7) mm, rotated rx 180 ry 0 rz -180 deg; joints [0, 0, 0, 0, 0, 0]
  Call Extruder 0.01786
  MoveL (T457) to (121.16, 113.02, 0.7) mm, rotated rx 180 ry 0 rz -180 deg; joints [0, 0, 0, 0, 0, 0]
  Call Extruder 0.39901
  MoveL (T458) to (111.98, 103.84, 0.7) mm, rotated rx 180 ry 0 rz -180 deg; joints [0, 0, 0, 0, 0, 0]
  Call Extruder 0.01786
  MoveL (T459) to (111.4, 103.84, 0.7) mm, rotated rx 180 ry 0 rz -180 deg; joints [0, 0, 0, 0, 0, 0]
  Call Extruder 0.42426
  MoveL (T460) to (121.16, 113.6, 0.7) mm, rotated rx 180 ry 0 rz -180 deg; joints [0, 0, 0, 0, 0, 0]
  Call Extruder 0.01786
  MoveL (T461) to (121.16, 114.19, 0.7) mm, rotated rx 180 ry 0 rz -180 deg; joints [0, 0, 0, 0, 0, 0]
  Call Extruder 0.44952
  MoveL (T462) to (110.81, 103.84, 0.7) mm, rotated rx 180 ry 0 rz -180 deg; joints [0, 0, 0, 0, 0, 0]
  Call Extruder 0.01786
  MoveL (T463) to (110.23, 103.84, 0.7) mm, rotated rx 180 ry 0 rz -180 deg; joints [0, 0, 0, 0, 0, 0]
  Call Extruder 0.47477
  MoveL (T464) to (121.16, 114.77, 0.7) mm, rotated rx 180 ry 0 rz -180 deg; joints [0, 0, 0, 0, 0, 0]
  Call Extruder 0.01786
  MoveL (T465) to (121.16, 115.35, 0.7) mm, rotated rx 180 ry 0 rz -180 deg; joints [0, 0, 0, 0, 0, 0]
  Call Extruder 0.50003
  MoveL (T466) to (109.65, 103.84, 0.7) mm, rotated rx 180 ry 0 rz -180 deg; joints [0, 0, 0, 0, 0, 0]
  Call Extruder 0.01786
  MoveL (T467) to (109.07, 103.84, 0.7) mm, rotated rx 180 ry 0 rz -180 deg; joints [0, 0, 0, 0, 0, 0]
  Call Extruder 0.52528
  MoveL (T468) to (121.16, 115.93, 0.7) mm, rotated rx 180 ry 0 rz -180 deg; joints [0, 0, 0, 0, 0, 0]
  Call Extruder 0.01786
  MoveL (T469) to (121.16, 116.51, 0.7) mm, rotated rx 180 ry 0 rz -180 deg; joints [0, 0, 0, 0, 0, 0]
  Call Extruder 0.55054
  MoveL (T470) to (108.49, 103.84, 0.7) mm, rotated rx 180 ry 0 rz -180 deg; joints [0, 0, 0, 0, 0, 0]
  Call Extruder 0.01786
  MoveL (T471) to (107.91, 103.84, 0.7) mm, rotated rx 180 ry 0 rz -180 deg; joints [0, 0, 0, 0, 0, 0]
  Call Extruder 0.57579
  MoveL (T472) to (121.16, 117.09, 0.7) mm, rotated rx 180 ry 0 rz -180 deg; joints [0, 0, 0, 0, 0, 0]
  Call Extruder 0.01786
  MoveL (T473) to (121.16, 117.67, 0.7) mm, rotated rx 180 ry 0 rz -180 deg; joints [0, 0, 0, 0, 0, 0]
  Call Extruder 0.60105
  MoveL (T474) to (107.33, 103.84, 0.7) mm, rotated rx 180 ry 0 rz -180 deg; joints [0, 0, 0, 0, 0, 0]
  Call Extruder 0.01786
  MoveL (T475) to (106.75, 103.84, 0.7) mm, rotated rx 180 ry 0 rz -180 deg; joints [0, 0, 0, 0, 0, 0]
  Call Extruder 0.6263
  MoveL (T476) to (121.16, 118.25, 0.7) mm, rotated rx 180 ry 0 rz -180 deg; joints [0, 0, 0, 0, 0, 0]
  Call Extruder 0.01786
  MoveL (T477) to (121.16, 118.83, 0.7) mm, rotated rx 180 ry 0 rz -180 deg; joints [0, 0, 0, 0, 0, 0]
  Call Extruder 0.65156
  MoveL (T478) to (106.17, 103.84, 0.7) mm, rotated rx 180 ry 0 rz -180 deg; joints [0, 0, 0, 0, 0, 0]
  Call Extruder 0.01786
  MoveL (T479) to (105.59, 103.84, 0.7) mm, rotated rx 180 ry 0 rz -180 deg; joints [0, 0, 0, 0, 0, 0]
  Call Extruder 0.67681
  MoveL (T480) to (121.16, 119.41, 0.7) mm, rotated rx 180 ry 0 rz -180 deg; joints [0, 0, 0, 0, 0, 0]
  Call Extruder 0.01786
  MoveL (T481) to (121.16, 119.99, 0.7) mm, rotated rx 180 ry 0 rz -180 deg; joints [0, 0, 0, 0, 0, 0]
  Call Extruder 0.70207
  MoveL (T482) to (105.01, 103.84, 0.7) mm, rotated rx 180 ry 0 rz -180 deg; joints [0, 0, 0, 0, 0, 0]
  Call Extruder 0.01786
  MoveL (T483) to (104.42, 103.84, 0.7) mm, rotated rx 180 ry 0 rz -180 deg; joints [0, 0, 0, 0, 0, 0]
  Call Extruder 0.72732
  MoveL (T484) to (121.16, 120.58, 0.7) mm, rotated rx 180 ry 0 rz -180 deg; joints [0, 0, 0, 0, 0, 0]
  Call Extruder 0.01786
  MoveL (T485) to (121.16, 121.16, 0.7) mm, rotated rx 180 ry 0 rz -180 deg; joints [0, 0, 0, 0, 0, 0]
  Call Extruder 0.75257
  MoveL (T486) to (103.84, 103.84, 0.7) mm, rotated rx 180 ry 0 rz -180 deg; joints [0, 0, 0, 0, 0, 0]
  Call Extruder 0.01786
  MoveL (T487) to (103.84, 104.42, 0.7) mm, rotated rx 180 ry 0 rz -180 deg; joints [0, 0, 0, 0, 0, 0]
  Call Extruder 0.72732
  MoveL (T488) to (120.58, 121.16, 0.7) mm, rotated rx 180 ry 0 rz -180 deg; joints [0, 0, 0, 0, 0, 0]
  Call Extruder 0.01786
  MoveL (T489) to (119.99, 121.16, 0.7) mm, rotated rx 180 ry 0 rz -180 deg; joints [0, 0, 0, 0, 0, 0]
  Call Extruder 0.70206
  MoveL (T490) to (103.84, 105.01, 0.7) mm, rotated rx 180 ry 0 rz -180 deg; joints [0, 0, 0, 0, 0, 0]
  Call Extruder 0.01786
  MoveL (T491) to (103.84, 105.59, 0.7) mm, rotated rx 180 ry 0 rz -180 deg; joints [0, 0, 0, 0, 0, 0]
  Call Extruder 0.67681
  MoveL (T492) to (119.41, 121.16, 0.7) mm, rotated rx 180 ry 0 rz -180 deg; joints [0, 0, 0, 0, 0, 0]
  Call Extruder 0.01786
  MoveL (T493) to (118.83, 121.16, 0.7) mm, rotated rx 180 ry 0 rz -180 deg; joints [0, 0, 0, 0, 0, 0]
  Call Extruder 0.65155
  MoveL (T494) to (103.84, 106.17, 0.7) mm, rotated rx 180 ry 0 rz -180 deg; joints [0, 0, 0, 0, 0, 0]
  Call Extruder 0.01786
  MoveL (T495) to (103.84, 106.75, 0.7) mm, rotated rx 180 ry 0 rz -180 deg; joints [0, 0, 0, 0, 0, 0]
  Call Extruder 0.6263
  MoveL (T496) to (118.25, 121.16, 0.7) mm, rotated rx 180 ry 0 rz -180 deg; joints [0, 0, 0, 0, 0, 0]
  Call Extruder 0.01786
  MoveL (T497) to (117.67, 121.16, 0.7) mm, rotated rx 180 ry 0 rz -180 deg; joints [0, 0, 0, 0, 0, 0]
  Call Extruder 0.60104
  MoveL (T498) to (103.84, 107.33, 0.7) mm, rotated rx 180 ry 0 rz -180 deg; joints [0, 0, 0, 0, 0, 0]
  Call Extruder 0.01786
  MoveL (T499) to (103.84, 107.91, 0.7) mm, rotated rx 180 ry 0 rz -180 deg; joints [0, 0, 0, 0, 0, 0]
  Call Extruder 0.57579
  MoveL (T500) to (117.09, 121.16, 0.7) mm, rotated rx 180 ry 0 rz -180 deg; joints [0, 0, 0, 0, 0, 0]
  Call Extruder 0.01786
  MoveL (T501) to (116.51, 121.16, 0.7) mm, rotated rx 180 ry 0 rz -180 deg; joints [0, 0, 0, 0, 0, 0]
  Call Extruder 0.55053
  MoveL (T502) to (103.84, 108.49, 0.7) mm, rotated rx 180 ry 0 rz -180 deg; joints [0, 0, 0, 0, 0, 0]
  Call Extruder 0.01786
  MoveL (T503) to (103.84, 109.07, 0.7) mm, rotated rx 180 ry 0 rz -180 deg; joints [0, 0, 0, 0, 0, 0]
  Call Extruder 0.52528
  MoveL (T504) to (115.93, 121.16, 0.7) mm, rotated rx 180 ry 0 rz -180 deg; joints [0, 0, 0, 0, 0, 0]
  Call Extruder 0.01786
  MoveL (T505) to (115.35, 121.16, 0.7) mm, rotated rx 180 ry 0 rz -180 deg; joints [0, 0, 0, 0, 0, 0]
  Call Extruder 0.50002
  MoveL (T506) to (103.84, 109.65, 0.7) mm, rotated rx 180 ry 0 rz -180 deg; joints [0, 0, 0, 0, 0, 0]
  Call Extruder 0.01786
  MoveL (T507) to (103.84, 110.23, 0.7) mm, rotated rx 180 ry 0 rz -180 deg; joints [0, 0, 0, 0, 0, 0]
  Call Extruder 0.47477
  MoveL (T508) to (114.77, 121.16, 0.7) mm, rotated rx 180 ry 0 rz -180 deg; joints [0, 0, 0, 0, 0, 0]
  Call Extruder 0.01786
  MoveL (T509) to (114.18, 121.16, 0.7) mm, rotated rx 180 ry 0 rz -180 deg; joints [0, 0, 0, 0, 0, 0]
  Call Extruder 0.44951
  MoveL (T510) to (103.84, 110.82, 0.7) mm, rotated rx 180 ry 0 rz -180 deg; joints [0, 0, 0, 0, 0, 0]
  Call Extruder 0.01786
  MoveL (T511) to (103.84, 111.4, 0.7) mm, rotated rx 180 ry 0 rz -180 deg; joints [0, 0, 0, 0, 0, 0]
  Call Extruder 0.42426
  MoveL (T512) to (113.6, 121.16, 0.7) mm, rotated rx 180 ry 0 rz -180 deg; joints [0, 0, 0, 0, 0, 0]
  Call Extruder 0.01786
  MoveL (T513) to (113.02, 121.16, 0.7) mm, rotated rx 180 ry 0 rz -180 deg; joints [0, 0, 0, 0, 0, 0]
  Call Extruder 0.399
  MoveL (T514) to (103.84, 111.98, 0.7) mm, rotated rx 180 ry 0 rz -180 deg; joints [0, 0, 0, 0, 0, 0]
  Call Extruder 0.01786
  MoveL (T515) to (103.84, 112.56, 0.7) mm, rotated rx 180 ry 0 rz -180 deg; joints [0, 0, 0, 0, 0, 0]
  Call Extruder 0.37375
  MoveL (T516) to (112.44, 121.16, 0.7) mm, rotated rx 180 ry 0 rz -180 deg; joints [0, 0, 0, 0, 0, 0]
  Call Extruder 0.01786
  MoveL (T517) to (111.86, 121.16, 0.7) mm, rotated rx 180 ry 0 rz -180 deg; joints [0, 0, 0, 0, 0, 0]
  Call Extruder 0.3485
  MoveL (T518) to (103.84, 113.14, 0.7) mm, rotated rx 180 ry 0 rz -180 deg; joints [0, 0, 0, 0, 0, 0]
  Call Extruder 0.01786
  MoveL (T519) to (103.84, 113.72, 0.7) mm, rotated rx 180 ry 0 rz -180 deg; joints [0, 0, 0, 0, 0, 0]
  Call Extruder 0.32324
  MoveL (T520) to (111.28, 121.16, 0.7) mm, rotated rx 180 ry 0 rz -180 deg; joints [0, 0, 0, 0, 0, 0]
  Call Extruder 0.01786
  MoveL (T521) to (110.7, 121.16, 0.7) mm, rotated rx 180 ry 0 rz -180 deg; joints [0, 0, 0, 0, 0, 0]
  Call Extruder 0.29799
  MoveL (T522) to (103.84, 114.3, 0.7) mm, rotated rx 180 ry 0 rz -180 deg; joints [0, 0, 0, 0, 0, 0]
  Call Extruder 0.01786
  MoveL (T523) to (103.84, 114.88, 0.7) mm, rotated rx 180 ry 0 rz -180 deg; joints [0, 0, 0, 0, 0, 0]
  Call Extruder 0.27273
  MoveL (T524) to (110.12, 121.16, 0.7) mm, rotated rx 180 ry 0 rz -180 deg; joints [0, 0, 0, 0, 0, 0]
  Call Extruder 0.01786
  MoveL (T525) to (109.54, 121.16, 0.7) mm, rotated rx 180 ry 0 rz -180 deg; joints [0, 0, 0, 0, 0, 0]
  Call Extruder 0.24748
  MoveL (T526) to (103.84, 115.46, 0.7) mm, rotated rx 180 ry 0 rz -180 deg; joints [0, 0, 0, 0, 0, 0]
  Call Extruder 0.01786
  MoveL (T527) to (103.84, 116.04, 0.7) mm, rotated rx 180 ry 0 rz -180 deg; joints [0, 0, 0, 0, 0, 0]
  Call Extruder 0.22222
  MoveL (T528) to (108.96, 121.16, 0.7) mm, rotated rx 180 ry 0 rz -180 deg; joints [0, 0, 0, 0, 0, 0]
  Call Extruder 0.01786
  MoveL (T529) to (108.38, 121.16, 0.7) mm, rotated rx 180 ry 0 rz -180 deg; joints [0, 0, 0, 0, 0, 0]
  Call Extruder 0.19697
  MoveL (T530) to (103.84, 116.62, 0.7) mm, rotated rx 180 ry 0 rz -180 deg; joints [0, 0, 0, 0, 0, 0]
  Call Extruder 0.01786
  MoveL (T531) to (103.84, 117.21, 0.7) mm, rotated rx 180 ry 0 rz -180 deg; joints [0, 0, 0, 0, 0, 0]
  Call Extruder 0.17171
  MoveL (T532) to (107.79, 121.16, 0.7) mm, rotated rx 180 ry 0 rz -180 deg; joints [0, 0, 0, 0, 0, 0]
  Call Extruder 0.01786
  MoveL (T533) to (107.21, 121.16, 0.7) mm, rotated rx 180 ry 0 rz -180 deg; joints [0, 0, 0, 0, 0, 0]
  Call Extruder 0.14646
  MoveL (T534) to (103.84, 117.79, 0.7) mm, rotated rx 180 ry 0 rz -180 deg; joints [0, 0, 0, 0, 0, 0]
  Call Extruder 0.01786
  MoveL (T535) to (103.84, 118.37, 0.7) mm, rotated rx 180 ry 0 rz -180 deg; joints [0, 0, 0, 0, 0, 0]
  Call Extruder 0.1212
  MoveL (T536) to (106.63, 121.16, 0.7) mm, rotated rx 180 ry 0 rz -180 deg; joints [0, 0, 0, 0, 0, 0]
  Call Extruder 0.01786
  MoveL (T537) to (106.05, 121.16, 0.7) mm, rotated rx 180 ry 0 rz -180 deg; joints [0, 0, 0, 0, 0, 0]
  Call Extruder 0.09595
  MoveL (T538) to (103.84, 118.95, 0.7) mm, rotated rx 180 ry 0 rz -180 deg; joints [0, 0, 0, 0, 0, 0]
  Call Extruder 0.01786
  MoveL (T539) to (103.84, 119.53, 0.7) mm, rotated rx 180 ry 0 rz -180 deg; joints [0, 0, 0, 0, 0, 0]
  Call Extruder 0.07069
  MoveL (T540) to (105.47, 121.16, 0.7) mm, rotated rx 180 ry 0 rz -180 deg; joints [0, 0, 0, 0, 0, 0]
  Call Extruder 0.01786
  MoveL (T541) to (104.89, 121.16, 0.7) mm, rotated rx 180 ry 0 rz -180 deg; joints [0, 0, 0, 0, 0, 0]
  Call Extruder 0.04544
  MoveL (T542) to (103.84, 120.11, 0.7) mm, rotated rx 180 ry 0 rz -180 deg; joints [0, 0, 0, 0, 0, 0]
  Call Extruder 0.01786
  MoveL (T543) to (103.84, 120.69, 0.7) mm, rotated rx 180 ry 0 rz -180 deg; joints [0, 0, 0, 0, 0, 0]
  Call Extruder 0.02815
  MoveL (T544) to (104.49, 121.34, 0.7) mm, rotated rx 180 ry 0 rz -180 deg; joints [0, 0, 0, 0, 0, 0]
  Call Extruder 0.02815
  Call Mcode M106 S255
  MoveL (T545) to (104.49, 121.34, 0.7) mm, rotated rx 180 ry 0 rz -180 deg; joints [0, 0, 0, 0, 0, 0]
  Set speed (45.0 mm/s)
  Call Extruder -1.6
  MoveL (T546) to (104.49, 121.34, 0.7) mm, rotated rx 180 ry 0 rz -180 deg; joints [0, 0, 0, 0, 0, 0]
  Set speed (120.0 mm/s)
  MoveL (T547) to (104.49, 121.34, 0.7) mm, rotated rx 180 ry 0 rz -180 deg; joints [0, 0, 0, 0, 0, 0]
  Call Extruder -0.3262
  MoveL (T548) to (103.84, 120.69, 0.7) mm, rotated rx 180 ry 0 rz -180 deg; joints [0, 0, 0, 0, 0, 0]
  Call Extruder -0.0538
  MoveL (T549) to (103.84, 120.54, 0.7) mm, rotated rx 180 ry 0 rz -180 deg; joints [0, 0, 0, 0, 0, 0]
  Set speed (45.0 mm/s)
  Call Extruder -0.02
  MoveL (T550) to (103.84, 120.54, 0.7) mm, rotated rx 180 ry 0 rz -180 deg; joints [0, 0, 0, 0, 0, 0]
  Set speed (150.0 mm/s)
  MoveL (T551) to (103.84, 120.54, 2.7) mm, rotated rx 180 ry 0 rz -180 deg; joints [0, 0, 0, 0, 0, 0]
  MoveL (T552) to (104.34, 103.54, 2.7) mm, rotated rx 180 ry 0 rz -180 deg; joints [0, 0, 0, 0, 0, 0]
  MoveL (T553) to (104.34, 103.54, 0.9) mm, rotated rx 180 ry 0 rz -180 deg; joints [0, 0, 0, 0, 0, 0]
  Set speed (40.0 mm/s)
  Call Extruder 2.0
  MoveL (T554) to (104.34, 103.54, 0.9) mm, rotated rx 180 ry 0 rz -180 deg; joints [0, 0, 0, 0, 0, 0]
  Call Extruder 0.52159
  MoveL (T555) to (121.46, 103.54, 0.9) mm, rotated rx 180 ry 0 rz -180 deg; joints [0, 0, 0, 0, 0, 0]
  Call Extruder 0.54596
  MoveL (T556) to (121.46, 121.46, 0.9) mm, rotated rx 180 ry 0 rz -180 deg; joints [0, 0, 0, 0, 0, 0]
  Call Extruder 0.54596
  MoveL (T557) to (103.54, 121.46, 0.9) mm, rotated rx 180 ry 0 rz -180 deg; joints [0, 0, 0, 0, 0, 0]
  Call Extruder 0.54596
  MoveL (T558) to (103.54, 103.54, 0.9) mm, rotated rx 180 ry 0 rz -180 deg; joints [0, 0, 0, 0, 0, 0]
  Call Extruder 0.02254
  MoveL (T559) to (104.28, 103.54, 0.9) mm, rotated rx 180 ry 0 rz -180 deg; joints [0, 0, 0, 0, 0, 0]
  Set speed (150.0 mm/s)
  MoveL (T560) to (103.53, 103.13, 0.9) mm, rotated rx 180 ry 0 rz -180 deg; joints [0, 0, 0, 0, 0, 0]
  Set speed (40.0 mm/s)
  MoveL (T561) to (103.53, 103.13, 0.9) mm, rotated rx 180 ry 0 rz -180 deg; joints [0, 0, 0, 0, 0, 0]
  Call Extruder 0.55858
  MoveL (T562) to (121.87, 103.13, 0.9) mm, rotated rx 180 ry 0 rz -180 deg; joints [0, 0, 0, 0, 0, 0]
  Call Extruder 0.57077
  MoveL (T563) to (121.87, 121.87, 0.9) mm, rotated rx 180 ry 0 rz -180 deg; joints [0, 0, 0, 0, 0, 0]
  Call Extruder 0.57077
  MoveL (T564) to (103.13, 121.87, 0.9) mm, rotated rx 180 ry 0 rz -180 deg; joints [0, 0, 0, 0, 0, 0]
  Call Extruder 0.57077
  MoveL (T565) to (103.13, 103.13, 0.9) mm, rotated rx 180 ry 0 rz -180 deg; joints [0, 0, 0, 0, 0, 0]
  Call Extruder 0.01036
  MoveL (T566) to (103.47, 103.13, 0.9) mm, rotated rx 180 ry 0 rz -180 deg; joints [0, 0, 0, 0, 0, 0]
  Set speed (150.0 mm/s)
  MoveL (T567) to (102.72, 102.81, 0.9) mm, rotated rx 180 ry 0 rz -180 deg; joints [0, 0, 0, 0, 0, 0]
  Set speed (25.0 mm/s)
  MoveL (T568) to (102.72, 102.81, 0.9) mm, rotated rx 180 ry 0 rz -180 deg; joints [0, 0, 0, 0, 0, 0]
  Call Extruder 0.00259
  MoveL (T569) to (102.72, 102.72, 0.9) mm, rotated rx 180 ry 0 rz -180 deg; joints [0, 0, 0, 0, 0, 0]
  Call Extruder 0.59557
  MoveL (T570) to (122.28, 102.72, 0.9) mm, rotated rx 180 ry 0 rz -180 deg; joints [0, 0, 0, 0, 0, 0]
  Call Extruder 0.59557
  MoveL (T571) to (122.28, 122.28, 0.9) mm, rotated rx 180 ry 0 rz -180 deg; joints [0, 0, 0, 0, 0, 0]
  Call Extruder 0.59557
  MoveL (T572) to (102.72, 122.28, 0.9) mm, rotated rx 180 ry 0 rz -180 deg; joints [0, 0, 0, 0, 0, 0]
  Call Extruder 0.59115
  MoveL (T573) to (102.72, 102.87, 0.9) mm, rotated rx 180 ry 0 rz -180 deg; joints [0, 0, 0, 0, 0, 0]
  Set speed (150.0 mm/s)
  MoveL (T574) to (102.78, 102.75, 0.9) mm, rotated rx 180 ry 0 rz -180 deg; joints [0, 0, 0, 0, 0, 0]
  Set speed (45.0 mm/s)
  Call Extruder -1.6
  MoveL (T575) to (102.78, 102.75, 0.9) mm, rotated rx 180 ry 0 rz -180 deg; joints [0, 0, 0, 0, 0, 0]
  Set speed (120.0 mm/s)
  MoveL (T576) to (102.78, 102.75, 0.9) mm, rotated rx 180 ry 0 rz -180 deg; joints [0, 0, 0, 0, 0, 0]
  Call Extruder -0.05166
  MoveL (T577) to (102.72, 102.72, 0.9) mm, rotated rx 180 ry 0 rz -180 deg; joints [0, 0, 0, 0, 0, 0]
  Call Extruder -0.32834
  MoveL (T578) to (103.65, 102.72, 0.9) mm, rotated rx 180 ry 0 rz -180 deg; joints [0, 0, 0, 0, 0, 0]
  Set speed (45.0 mm/s)
  Call Extruder -0.02
  MoveL (T579) to (103.65, 102.72, 0.9) mm, rotated rx 180 ry 0 rz -180 deg; joints [0, 0, 0, 0, 0, 0]
  Set speed (150.0 mm/s)
  MoveL (T580) to (103.65, 102.72, 2.9) mm, rotated rx 180 ry 0 rz -180 deg; joints [0, 0, 0, 0, 0, 0]
  MoveL (T581) to (121.34, 120.51, 2.9) mm, rotated rx 180 ry 0 rz -180 deg; joints [0, 0, 0, 0, 0, 0]
  MoveL (T582) to (121.34, 120.51, 0.9) mm, rotated rx 180 ry 0 rz -180 deg; joints [0, 0, 0, 0, 0, 0]
  Set speed (40.0 mm/s)
  Call Extruder 2.0
  MoveL (T583) to (121.34, 120.51, 0.9) mm, rotated rx 180 ry 0 rz -180 deg; joints [0, 0, 0, 0, 0, 0]
  Call Extruder 0.02815
  MoveL (T584) to (120.69, 121.16, 0.9) mm, rotated rx 180 ry 0 rz -180 deg; joints [0, 0, 0, 0, 0, 0]
  Call Extruder 0.01786
  MoveL (T585) to (120.11, 121.16, 0.9) mm, rotated rx 180 ry 0 rz -180 deg; joints [0, 0, 0, 0, 0, 0]
  Call Extruder 0.04544
  MoveL (T586) to (121.16, 120.11, 0.9) mm, rotated rx 180 ry 0 rz -180 deg; joints [0, 0, 0, 0, 0, 0]
  Call Extruder 0.01786
  MoveL (T587) to (121.16, 119.53, 0.9) mm, rotated rx 180 ry 0 rz -180 deg; joints [0, 0, 0, 0, 0, 0]
  Call Extruder 0.0707
  MoveL (T588) to (119.53, 121.16, 0.9) mm, rotated rx 180 ry 0 rz -180 deg; joints [0, 0, 0, 0, 0, 0]
  Call Extruder 0.01786
  MoveL (T589) to (118.95, 121.16, 0.9) mm, rotated rx 180 ry 0 rz -180 deg; joints [0, 0, 0, 0, 0, 0]
  Call Extruder 0.09595
  MoveL (T590) to (121.16, 118.95, 0.9) mm, rotated rx 180 ry 0 rz -180 deg; joints [0, 0, 0, 0, 0, 0]
  Call Extruder 0.01786
  MoveL (T591) to (121.16, 118.37, 0.9) mm, rotated rx 180 ry 0 rz -180 deg; joints [0, 0, 0, 0, 0, 0]
  Call Extruder 0.12121
  MoveL (T592) to (118.37, 121.16, 0.9) mm, rotated rx 180 ry 0 rz -180 deg; joints [0, 0, 0, 0, 0, 0]
  Call Extruder 0.01786
  MoveL (T593) to (117.79, 121.16, 0.9) mm, rotated rx 180 ry 0 rz -180 deg; joints [0, 0, 0, 0, 0, 0]
  Call Extruder 0.14646
  MoveL (T594) to (121.16, 117.79, 0.9) mm, rotated rx 180 ry 0 rz -180 deg; joints [0, 0, 0, 0, 0, 0]
  Call Extruder 0.01786
  MoveL (T595) to (121.16, 117.21, 0.9) mm, rotated rx 180 ry 0 rz -180 deg; joints [0, 0, 0, 0, 0, 0]
  Call Extruder 0.17172
  MoveL (T596) to (117.21, 121.16, 0.9) mm, rotated rx 180 ry 0 rz -180 deg; joints [0, 0, 0, 0, 0, 0]
  Call Extruder 0.01786
  MoveL (T597) to (116.62, 121.16, 0.9) mm, rotated rx 180 ry 0 rz -180 deg; joints [0, 0, 0, 0, 0, 0]
  Call Extruder 0.19697
  MoveL (T598) to (121.16, 116.62, 0.9) mm, rotated rx 180 ry 0 rz -180 deg; joints [0, 0, 0, 0, 0, 0]
  Call Extruder 0.01786
  MoveL (T599) to (121.16, 116.04, 0.9) mm, rotated rx 180 ry 0 rz -180 deg; joints [0, 0, 0, 0, 0, 0]
  Call Extruder 0.22223
  MoveL (T600) to (116.04, 121.16, 0.9) mm, rotated rx 180 ry 0 rz -180 deg; joints [0, 0, 0, 0, 0, 0]
  Call Extruder 0.01786
  MoveL (T601) to (115.46, 121.16, 0.9) mm, rotated rx 180 ry 0 rz -180 deg; joints [0, 0, 0, 0, 0, 0]
  Call Extruder 0.24748
  MoveL (T602) to (121.16, 115.46, 0.9) mm, rotated rx 180 ry 0 rz -180 deg; joints [0, 0, 0, 0, 0, 0]
  Call Extruder 0.01786
  MoveL (T603) to (121.16, 114.88, 0.9) mm, rotated rx 180 ry 0 rz -180 deg; joints [0, 0, 0, 0, 0, 0]
  Call Extruder 0.27274
  MoveL (T604) to (114.88, 121.16, 0.9) mm, rotated rx 180 ry 0 rz -180 deg; joints [0, 0, 0, 0, 0, 0]
  Call Extruder 0.01786
  MoveL (T605) to (114.3, 121.16, 0.9) mm, rotated rx 180 ry 0 rz -180 deg; joints [0, 0, 0, 0, 0, 0]
  Call Extruder 0.29799
  MoveL (T606) to (121.16, 114.3, 0.9) mm, rotated rx 180 ry 0 rz -180 deg; joints [0, 0, 0, 0, 0, 0]
  Call Extruder 0.01786
  MoveL (T607) to (121.16, 113.72, 0.9) mm, rotated rx 180 ry 0 rz -180 deg; joints [0, 0, 0, 0, 0, 0]
  Call Extruder 0.32324
  MoveL (T608) to (113.72, 121.16, 0.9) mm, rotated rx 180 ry 0 rz -180 deg; joints [0, 0, 0, 0, 0, 0]
  Call Extruder 0.01786
  MoveL (T609) to (113.14, 121.16, 0.9) mm, rotated rx 180 ry 0 rz -180 deg; joints [0, 0, 0, 0, 0, 0]
  Call Extruder 0.3485
  MoveL (T610) to (121.16, 113.14, 0.9) mm, rotated rx 180 ry 0 rz -180 deg; joints [0, 0, 0, 0, 0, 0]
  Call Extruder 0.01786
  MoveL (T611) to (121.16, 112.56, 0.9) mm, rotated rx 180 ry 0 rz -180 deg; joints [0, 0, 0, 0, 0, 0]
  Call Extruder 0.37375
  MoveL (T612) to (112.56, 121.16, 0.9) mm, rotated rx 180 ry 0 rz -180 deg; joints [0, 0, 0, 0, 0, 0]
  Call Extruder 0.01786
  MoveL (T613) to (111.98, 121.16, 0.9) mm, rotated rx 180 ry 0 rz -180 deg; joints [0, 0, 0, 0, 0, 0]
  Call Extruder 0.39901
  MoveL (T614) to (121.16, 111.98, 0.9) mm, rotated rx 180 ry 0 rz -180 deg; joints [0, 0, 0, 0, 0, 0]
  Call Extruder 0.01786
  MoveL (T615) to (121.16, 111.4, 0.9) mm, rotated rx 180 ry 0 rz -180 deg; joints [0, 0, 0, 0, 0, 0]
  Call Extruder 0.42426
  MoveL (T616) to (111.4, 121.16, 0.9) mm, rotated rx 180 ry 0 rz -180 deg; joints [0, 0, 0, 0, 0, 0]
  Call Extruder 0.01786
  MoveL (T617) to (110.81, 121.16, 0.9) mm, rotated rx 180 ry 0 rz -180 deg; joints [0, 0, 0, 0, 0, 0]
  Call Extruder 0.44952
  MoveL (T618) to (121.16, 110.81, 0.9) mm, rotated rx 180 ry 0 rz -180 deg; joints [0, 0, 0, 0, 0, 0]
  Call Extruder 0.01786
  MoveL (T619) to (121.16, 110.23, 0.9) mm, rotated rx 180 ry 0 rz -180 deg; joints [0, 0, 0, 0, 0, 0]
  Call Extruder 0.47477
  MoveL (T620) to (110.23, 121.16, 0.9) mm, rotated rx 180 ry 0 rz -180 deg; joints [0, 0, 0, 0, 0, 0]
  Call Extruder 0.01786
  MoveL (T621) to (109.65, 121.16, 0.9) mm, rotated rx 180 ry 0 rz -180 deg; joints [0, 0, 0, 0, 0, 0]
  Call Extruder 0.50003
  MoveL (T622) to (121.16, 109.65, 0.9) mm, rotated rx 180 ry 0 rz -180 deg; joints [0, 0, 0, 0, 0, 0]
  Call Extruder 0.01786
  MoveL (T623) to (121.16, 109.07, 0.9) mm, rotated rx 180 ry 0 rz -180 deg; joints [0, 0, 0, 0, 0, 0]
  Call Extruder 0.52528
  MoveL (T624) to (109.07, 121.16, 0.9) mm, rotated rx 180 ry 0 rz -180 deg; joints [0, 0, 0, 0, 0, 0]
  Call Extruder 0.01786
  MoveL (T625) to (108.49, 121.16, 0.9) mm, rotated rx 180 ry 0 rz -180 deg; joints [0, 0, 0, 0, 0, 0]
  Call Extruder 0.55054
  MoveL (T626) to (121.16, 108.49, 0.9) mm, rotated rx 180 ry 0 rz -180 deg; joints [0, 0, 0, 0, 0, 0]
  Call Extruder 0.01786
  MoveL (T627) to (121.16, 107.91, 0.9) mm, rotated rx 180 ry 0 rz -180 deg; joints [0, 0, 0, 0, 0, 0]
  Call Extruder 0.57579
  MoveL (T628) to (107.91, 121.16, 0.9) mm, rotated rx 180 ry 0 rz -180 deg; joints [0, 0, 0, 0, 0, 0]
  Call Extruder 0.01786
  MoveL (T629) to (107.33, 121.16, 0.9) mm, rotated rx 180 ry 0 rz -180 deg; joints [0, 0, 0, 0, 0, 0]
  Call Extruder 0.60105
  MoveL (T630) to (121.16, 107.33, 0.9) mm, rotated rx 180 ry 0 rz -180 deg; joints [0, 0, 0, 0, 0, 0]
  Call Extruder 0.01786
  MoveL (T631) to (121.16, 106.75, 0.9) mm, rotated rx 180 ry 0 rz -180 deg; joints [0, 0, 0, 0, 0, 0]
  Call Extruder 0.6263
  MoveL (T632) to (106.75, 121.16, 0.9) mm, rotated rx 180 ry 0 rz -180 deg; joints [0, 0, 0, 0, 0, 0]
  Call Extruder 0.01786
  MoveL (T633) to (106.17, 121.16, 0.9) mm, rotated rx 180 ry 0 rz -180 deg; joints [0, 0, 0, 0, 0, 0]
  Call Extruder 0.65156
  MoveL (T634) to (121.16, 106.17, 0.9) mm, rotated rx 180 ry 0 rz -180 deg; joints [0, 0, 0, 0, 0, 0]
  Call Extruder 0.01786
  MoveL (T635) to (121.16, 105.59, 0.9) mm, rotated rx 180 ry 0 rz -180 deg; joints [0, 0, 0, 0, 0, 0]
  Call Extruder 0.67681
  MoveL (T636) to (105.59, 121.16, 0.9) mm, rotated rx 180 ry 0 rz -180 deg; joints [0, 0, 0, 0, 0, 0]
  Call Extruder 0.01786
  MoveL (T637) to (105.01, 121.16, 0.9) mm, rotated rx 180 ry 0 rz -180 deg; joints [0, 0, 0, 0, 0, 0]
  Call Extruder 0.70207
  MoveL (T638) to (121.16, 105.01, 0.9) mm, rotated rx 180 ry 0 rz -180 deg; joints [0, 0, 0, 0, 0, 0]
  Call Extruder 0.01786
  MoveL (T639) to (121.16, 104.42, 0.9) mm, rotated rx 180 ry 0 rz -180 deg; joints [0, 0, 0, 0, 0, 0]
  Call Extruder 0.72732
  MoveL (T640) to (104.42, 121.16, 0.9) mm, rotated rx 180 ry 0 rz -180 deg; joints [0, 0, 0, 0, 0, 0]
  Call Extruder 0.01786
  MoveL (T641) to (103.84, 121.16, 0.9) mm, rotated rx 180 ry 0 rz -180 deg; joints [0, 0, 0, 0, 0, 0]
  Call Extruder 0.75257
  MoveL (T642) to (121.16, 103.84, 0.9) mm, rotated rx 180 ry 0 rz -180 deg; joints [0, 0, 0, 0, 0, 0]
  Call Extruder 0.01786
  MoveL (T643) to (120.58, 103.84, 0.9) mm, rotated rx 180 ry 0 rz -180 deg; joints [0, 0, 0, 0, 0, 0]
  Call Extruder 0.72732
  MoveL (T644) to (103.84, 120.58, 0.9) mm, rotated rx 180 ry 0 rz -180 deg; joints [0, 0, 0, 0, 0, 0]
  Call Extruder 0.01786
  MoveL (T645) to (103.84, 119.99, 0.9) mm, rotated rx 180 ry 0 rz -180 deg; joints [0, 0, 0, 0, 0, 0]
  Call Extruder 0.70206
  MoveL (T646) to (119.99, 103.84, 0.9) mm, rotated rx 180 ry 0 rz -180 deg; joints [0, 0, 0, 0, 0, 0]
  Call Extruder 0.01786
  MoveL (T647) to (119.41, 103.84, 0.9) mm, rotated rx 180 ry 0 rz -180 deg; joints [0, 0, 0, 0, 0, 0]
  Call Extruder 0.67681
  MoveL (T648) to (103.84, 119.41, 0.9) mm, rotated rx 180 ry 0 rz -180 deg; joints [0, 0, 0, 0, 0, 0]
  Call Extruder 0.01786
  MoveL (T649) to (103.84, 118.83, 0.9) mm, rotated rx 180 ry 0 rz -180 deg; joints [0, 0, 0, 0, 0, 0]
  Call Extruder 0.65155
  MoveL (T650) to (118.83, 103.84, 0.9) mm, rotated rx 180 ry 0 rz -180 deg; joints [0, 0, 0, 0, 0, 0]
  Call Extruder 0.01786
  MoveL (T651) to (118.25, 103.84, 0.9) mm, rotated rx 180 ry 0 rz -180 deg; joints [0, 0, 0, 0, 0, 0]
  Call Extruder 0.6263
  MoveL (T652) to (103.84, 118.25, 0.9) mm, rotated rx 180 ry 0 rz -180 deg; joints [0, 0, 0, 0, 0, 0]
  Call Extruder 0.01786
  MoveL (T653) to (103.84, 117.67, 0.9) mm, rotated rx 180 ry 0 rz -180 deg; joints [0, 0, 0, 0, 0, 0]
  Call Extruder 0.60104
  MoveL (T654) to (117.67, 103.84, 0.9) mm, rotated rx 180 ry 0 rz -180 deg; joints [0, 0, 0, 0, 0, 0]
  Call Extruder 0.01786
  MoveL (T655) to (117.09, 103.84, 0.9) mm, rotated rx 180 ry 0 rz -180 deg; joints [0, 0, 0, 0, 0, 0]
  Call Extruder 0.57579
  MoveL (T656) to (103.84, 117.09, 0.9) mm, rotated rx 180 ry 0 rz -180 deg; joints [0, 0, 0, 0, 0, 0]
  Call Extruder 0.01786
  MoveL (T657) to (103.84, 116.51, 0.9) mm, rotated rx 180 ry 0 rz -180 deg; joints [0, 0, 0, 0, 0, 0]
  Call Extruder 0.55053
  MoveL (T658) to (116.51, 103.84, 0.9) mm, rotated rx 180 ry 0 rz -180 deg; joints [0, 0, 0, 0, 0, 0]
  Call Extruder 0.01786
  MoveL (T659) to (115.93, 103.84, 0.9) mm, rotated rx 180 ry 0 rz -180 deg; joints [0, 0, 0, 0, 0, 0]
  Call Extruder 0.52528
  MoveL (T660) to (103.84, 115.93, 0.9) mm, rotated rx 180 ry 0 rz -180 deg; joints [0, 0, 0, 0, 0, 0]
  Call Extruder 0.01786
  MoveL (T661) to (103.84, 115.35, 0.9) mm, rotated rx 180 ry 0 rz -180 deg; joints [0, 0, 0, 0, 0, 0]
  Call Extruder 0.50002
  MoveL (T662) to (115.35, 103.84, 0.9) mm, rotated rx 180 ry 0 rz -180 deg; joints [0, 0, 0, 0, 0, 0]
  Call Extruder 0.01786
  MoveL (T663) to (114.77, 103.84, 0.9) mm, rotated rx 180 ry 0 rz -180 deg; joints [0, 0, 0, 0, 0, 0]
  Call Extruder 0.47477
  MoveL (T664) to (103.84, 114.77, 0.9) mm, rotated rx 180 ry 0 rz -180 deg; joints [0, 0, 0, 0, 0, 0]
  Call Extruder 0.01786
  MoveL (T665) to (103.84, 114.18, 0.9) mm, rotated rx 180 ry 0 rz -180 deg; joints [0, 0, 0, 0, 0, 0]
  Call Extruder 0.44951
  MoveL (T666) to (114.18, 103.84, 0.9) mm, rotated rx 180 ry 0 rz -180 deg; joints [0, 0, 0, 0, 0, 0]
  Call Extruder 0.01786
  MoveL (T667) to (113.6, 103.84, 0.9) mm, rotated rx 180 ry 0 rz -180 deg; joints [0, 0, 0, 0, 0, 0]
  Call Extruder 0.42426
  MoveL (T668) to (103.84, 113.6, 0.9) mm, rotated rx 180 ry 0 rz -180 deg; joints [0, 0, 0, 0, 0, 0]
  Call Extruder 0.01786
  MoveL (T669) to (103.84, 113.02, 0.9) mm, rotated rx 180 ry 0 rz -180 deg; joints [0, 0, 0, 0, 0, 0]
  Call Extruder 0.399
  MoveL (T670) to (113.02, 103.84, 0.9) mm, rotated rx 180 ry 0 rz -180 deg; joints [0, 0, 0, 0, 0, 0]
  Call Extruder 0.01786
  MoveL (T671) to (112.44, 103.84, 0.9) mm, rotated rx 180 ry 0 rz -180 deg; joints [0, 0, 0, 0, 0, 0]
  Call Extruder 0.37375
  MoveL (T672) to (103.84, 112.44, 0.9) mm, rotated rx 180 ry 0 rz -180 deg; joints [0, 0, 0, 0, 0, 0]
  Call Extruder 0.01786
  MoveL (T673) to (103.84, 111.86, 0.9) mm, rotated rx 180 ry 0 rz -180 deg; joints [0, 0, 0, 0, 0, 0]
  Call Extruder 0.3485
  MoveL (T674) to (111.86, 103.84, 0.9) mm, rotated rx 180 ry 0 rz -180 deg; joints [0, 0, 0, 0, 0, 0]
  Call Extruder 0.01786
  MoveL (T675) to (111.28, 103.84, 0.9) mm, rotated rx 180 ry 0 rz -180 deg; joints [0, 0, 0, 0, 0, 0]
  Call Extruder 0.32324
  MoveL (T676) to (103.84, 111.28, 0.9) mm, rotated rx 180 ry 0 rz -180 deg; joints [0, 0, 0, 0, 0, 0]
  Call Extruder 0.01786
  MoveL (T677) to (103.84, 110.7, 0.9) mm, rotated rx 180 ry 0 rz -180 deg; joints [0, 0, 0, 0, 0, 0]
  Call Extruder 0.29799
  MoveL (T678) to (110.7, 103.84, 0.9) mm, rotated rx 180 ry 0 rz -180 deg; joints [0, 0, 0, 0, 0, 0]
  Call Extruder 0.01786
  MoveL (T679) to (110.12, 103.84, 0.9) mm, rotated rx 180 ry 0 rz -180 deg; joints [0, 0, 0, 0, 0, 0]
  Call Extruder 0.27273
  MoveL (T680) to (103.84, 110.12, 0.9) mm, rotated rx 180 ry 0 rz -180 deg; joints [0, 0, 0, 0, 0, 0]
  Call Extruder 0.01786
  MoveL (T681) to (103.84, 109.54, 0.9) mm, rotated rx 180 ry 0 rz -180 deg; joints [0, 0, 0, 0, 0, 0]
  Call Extruder 0.24748
  MoveL (T682) to (109.54, 103.84, 0.9) mm, rotated rx 180 ry 0 rz -180 deg; joints [0, 0, 0, 0, 0, 0]
  Call Extruder 0.01786
  MoveL (T683) to (108.96, 103.84, 0.9) mm, rotated rx 180 ry 0 rz -180 deg; joints [0, 0, 0, 0, 0, 0]
  Call Extruder 0.22222
  MoveL (T684) to (103.84, 108.96, 0.9) mm, rotated rx 180 ry 0 rz -180 deg; joints [0, 0, 0, 0, 0, 0]
  Call Extruder 0.01786
  MoveL (T685) to (103.84, 108.38, 0.9) mm, rotated rx 180 ry 0 rz -180 deg; joints [0, 0, 0, 0, 0, 0]
  Call Extruder 0.19697
  MoveL (T686) to (108.38, 103.84, 0.9) mm, rotated rx 180 ry 0 rz -180 deg; joints [0, 0, 0, 0, 0, 0]
  Call Extruder 0.01786
  MoveL (T687) to (107.79, 103.84, 0.9) mm, rotated rx 180 ry 0 rz -180 deg; joints [0, 0, 0, 0, 0, 0]
  Call Extruder 0.17171
  MoveL (T688) to (103.84, 107.79, 0.9) mm, rotated rx 180 ry 0 rz -180 deg; joints [0, 0, 0, 0, 0, 0]
  Call Extruder 0.01786
  MoveL (T689) to (103.84, 107.21, 0.9) mm, rotated rx 180 ry 0 rz -180 deg; joints [0, 0, 0, 0, 0, 0]
  Call Extruder 0.14646
  MoveL (T690) to (107.21, 103.84, 0.9) mm, rotated rx 180 ry 0 rz -180 deg; joints [0, 0, 0, 0, 0, 0]
  Call Extruder 0.01786
  MoveL (T691) to (106.63, 103.84, 0.9) mm, rotated rx 180 ry 0 rz -180 deg; joints [0, 0, 0, 0, 0, 0]
  Call Extruder 0.1212
  MoveL (T692) to (103.84, 106.63, 0.9) mm, rotated rx 180 ry 0 rz -180 deg; joints [0, 0, 0, 0, 0, 0]
  Call Extruder 0.01786
  MoveL (T693) to (103.84, 106.05, 0.9) mm, rotated rx 180 ry 0 rz -180 deg; joints [0, 0, 0, 0, 0, 0]
  Call Extruder 0.09595
  MoveL (T694) to (106.05, 103.84, 0.9) mm, rotated rx 180 ry 0 rz -180 deg; joints [0, 0, 0, 0, 0, 0]
  Call Extruder 0.01786
  MoveL (T695) to (105.47, 103.84, 0.9) mm, rotated rx 180 ry 0 rz -180 deg; joints [0, 0, 0, 0, 0, 0]
  Call Extruder 0.07069
  MoveL (T696) to (103.84, 105.47, 0.9) mm, rotated rx 180 ry 0 rz -180 deg; joints [0, 0, 0, 0, 0, 0]
  Call Extruder 0.01786
  MoveL (T697) to (103.84, 104.89, 0.9) mm, rotated rx 180 ry 0 rz -180 deg; joints [0, 0, 0, 0, 0, 0]
  Call Extruder 0.04544
  MoveL (T698) to (104.89, 103.84, 0.9) mm, rotated rx 180 ry 0 rz -180 deg; joints [0, 0, 0, 0, 0, 0]
  Call Extruder 0.01786
  MoveL (T699) to (104.31, 103.84, 0.9) mm, rotated rx 180 ry 0 rz -180 deg; joints [0, 0, 0, 0, 0, 0]
  Call Extruder 0.02815
  MoveL (T700) to (103.66, 104.49, 0.9) mm, rotated rx 180 ry 0 rz -180 deg; joints [0, 0, 0, 0, 0, 0]
  Set speed (45.0 mm/s)
  Call Extruder -1.6
  MoveL (T701) to (103.66, 104.49, 0.9) mm, rotated rx 180 ry 0 rz -180 deg; joints [0, 0, 0, 0, 0, 0]
  Set speed (120.0 mm/s)
  MoveL (T702) to (103.66, 104.49, 0.9) mm, rotated rx 180 ry 0 rz -180 deg; joints [0, 0, 0, 0, 0, 0]
  Call Extruder -0.3262
  MoveL (T703) to (104.31, 103.84, 0.9) mm, rotated rx 180 ry 0 rz -180 deg; joints [0, 0, 0, 0, 0, 0]
  Call Extruder -0.0538
  MoveL (T704) to (104.46, 103.84, 0.9) mm, rotated rx 180 ry 0 rz -180 deg; joints [0, 0, 0, 0, 0, 0]
  Set speed (45.0 mm/s)
  Call Extruder -0.02
  MoveL (T705) to (104.46, 103.84, 0.9) mm, rotated rx 180 ry 0 rz -180 deg; joints [0, 0, 0, 0, 0, 0]
  Set speed (150.0 mm/s)
  MoveL (T706) to (104.46, 103.84, 2.9) mm, rotated rx 180 ry 0 rz -180 deg; joints [0, 0, 0, 0, 0, 0]
  MoveL (T707) to (104.34, 103.54, 2.9) mm, rotated rx 180 ry 0 rz -180 deg; joints [0, 0, 0, 0, 0, 0]
  MoveL (T708) to (104.34, 103.54, 1.1) mm, rotated rx 180 ry 0 rz -180 deg; joints [0, 0, 0, 0, 0, 0]
  Set speed (40.0 mm/s)
  Call Extruder 2.0
  MoveL (T709) to (104.34, 103.54, 1.1) mm, rotated rx 180 ry 0 rz -180 deg; joints [0, 0, 0, 0, 0, 0]
  Call Extruder 0.52159
  MoveL (T710) to (121.46, 103.54, 1.1) mm, rotated rx 180 ry 0 rz -180 deg; joints [0, 0, 0, 0, 0, 0]
  Call Extruder 0.54596
  MoveL (T711) to (121.46, 121.46, 1.1) mm, rotated rx 180 ry 0 rz -180 deg; joints [0, 0, 0, 0, 0, 0]
  Call Extruder 0.54596
  MoveL (T712) to (103.54, 121.46, 1.1) mm, rotated rx 180 ry 0 rz -180 deg; joints [0, 0, 0, 0, 0, 0]
  Call Extruder 0.54596
  MoveL (T713) to (103.54, 103.54, 1.1) mm, rotated rx 180 ry 0 rz -180 deg; joints [0, 0, 0, 0, 0, 0]
  Call Extruder 0.02254
  MoveL (T714) to (104.28, 103.54, 1.1) mm, rotated rx 180 ry 0 rz -180 deg; joints [0, 0, 0, 0, 0, 0]
  Set speed (150.0 mm/s)
  MoveL (T715) to (103.53, 103.13, 1.1) mm, rotated rx 180 ry 0 rz -180 deg; joints [0, 0, 0, 0, 0, 0]
  Set speed (40.0 mm/s)
  MoveL (T716) to (103.53, 103.13, 1.1) mm, rotated rx 180 ry 0 rz -180 deg; joints [0, 0, 0, 0, 0, 0]
  Call Extruder 0.55858
  MoveL (T717) to (121.87, 103.13, 1.1) mm, rotated rx 180 ry 0 rz -180 deg; joints [0, 0, 0, 0, 0, 0]
  Call Extruder 0.57077
  MoveL (T718) to (121.87, 121.87, 1.1) mm, rotated rx 180 ry 0 rz -180 deg; joints [0, 0, 0, 0, 0, 0]
  Call Extruder 0.57077
  MoveL (T719) to (103.13, 121.87, 1.1) mm, rotated rx 180 ry 0 rz -180 deg; joints [0, 0, 0, 0, 0, 0]
  Call Extruder 0.57077
  MoveL (T720) to (103.13, 103.13, 1.1) mm, rotated rx 180 ry 0 rz -180 deg; joints [0, 0, 0, 0, 0, 0]
  Call Extruder 0.01036
  MoveL (T721) to (103.47, 103.13, 1.1) mm, rotated rx 180 ry 0 rz -180 deg; joints [0, 0, 0, 0, 0, 0]
  Set speed (150.0 mm/s)
  MoveL (T722) to (102.72, 102.81, 1.1) mm, rotated rx 180 ry 0 rz -180 deg; joints [0, 0, 0, 0, 0, 0]
  Set speed (25.0 mm/s)
  MoveL (T723) to (102.72, 102.81, 1.1) mm, rotated rx 180 ry 0 rz -180 deg; joints [0, 0, 0, 0, 0, 0]
  Call Extruder 0.00259
  MoveL (T724) to (102.72, 102.72, 1.1) mm, rotated rx 180 ry 0 rz -180 deg; joints [0, 0, 0, 0, 0, 0]
  Call Extruder 0.59557
  MoveL (T725) to (122.28, 102.72, 1.1) mm, rotated rx 180 ry 0 rz -180 deg; joints [0, 0, 0, 0, 0, 0]
  Call Extruder 0.59557
  MoveL (T726) to (122.28, 122.28, 1.1) mm, rotated rx 180 ry 0 rz -180 deg; joints [0, 0, 0, 0, 0, 0]
  Call Extruder 0.59557
  MoveL (T727) to (102.72, 122.28, 1.1) mm, rotated rx 180 ry 0 rz -180 deg; joints [0, 0, 0, 0, 0, 0]
  Call Extruder 0.59115
  MoveL (T728) to (102.72, 102.87, 1.1) mm, rotated rx 180 ry 0 rz -180 deg; joints [0, 0, 0, 0, 0, 0]
  Set speed (150.0 mm/s)
  MoveL (T729) to (102.78, 102.75, 1.1) mm, rotated rx 180 ry 0 rz -180 deg; joints [0, 0, 0, 0, 0, 0]
  Set speed (45.0 mm/s)
  Call Extruder -1.6
  MoveL (T730) to (102.78, 102.75, 1.1) mm, rotated rx 180 ry 0 rz -180 deg; joints [0, 0, 0, 0, 0, 0]
  Set speed (120.0 mm/s)
  MoveL (T731) to (102.78, 102.75, 1.1) mm, rotated rx 180 ry 0 rz -180 deg; joints [0, 0, 0, 0, 0, 0]
  Call Extruder -0.05166
  MoveL (T732) to (102.72, 102.72, 1.1) mm, rotated rx 180 ry 0 rz -180 deg; joints [0, 0, 0, 0, 0, 0]
  Call Extruder -0.32834
  MoveL (T733) to (103.65, 102.72, 1.1) mm, rotated rx 180 ry 0 rz -180 deg; joints [0, 0, 0, 0, 0, 0]
  Set speed (45.0 mm/s)
  Call Extruder -0.02
  MoveL (T734) to (103.65, 102.72, 1.1) mm, rotated rx 180 ry 0 rz -180 deg; joints [0, 0, 0, 0, 0, 0]
  Set speed (150.0 mm/s)
  MoveL (T735) to (103.65, 102.72, 3.1) mm, rotated rx 180 ry 0 rz -180 deg; joints [0, 0, 0, 0, 0, 0]
  MoveL (T736) to (120.51, 103.66, 3.1) mm, rotated rx 180 ry 0 rz -180 deg; joints [0, 0, 0, 0, 0, 0]
  MoveL (T737) to (120.51, 103.66, 1.1) mm, rotated rx 180 ry 0 rz -180 deg; joints [0, 0, 0, 0, 0, 0]
  Set speed (40.0 mm/s)
  Call Extruder 2.0
  MoveL (T738) to (120.51, 103.66, 1.1) mm, rotated rx 180 ry 0 rz -180 deg; joints [0, 0, 0, 0, 0, 0]
  Call Extruder 0.02815
  MoveL (T739) to (121.16, 104.31, 1.1) mm, rotated rx 180 ry 0 rz -180 deg; joints [0, 0, 0, 0, 0, 0]
  Call Extruder 0.01786
  MoveL (T740) to (121.16, 104.89, 1.1) mm, rotated rx 180 ry 0 rz -180 deg; joints [0, 0, 0, 0, 0, 0]
  Call Extruder 0.04544
  MoveL (T741) to (120.11, 103.84, 1.1) mm, rotated rx 180 ry 0 rz -180 deg; joints [0, 0, 0, 0, 0, 0]
  Call Extruder 0.01786
  MoveL (T742) to (119.53, 103.84, 1.1) mm, rotated rx 180 ry 0 rz -180 deg; joints [0, 0, 0, 0, 0, 0]
  Call Extruder 0.0707
  MoveL (T743) to (121.16, 105.47, 1.1) mm, rotated rx 180 ry 0 rz -180 deg; joints [0, 0, 0, 0, 0, 0]
  Call Extruder 0.01786
  MoveL (T744) to (121.16, 106.05, 1.1) mm, rotated rx 180 ry 0 rz -180 deg; joints [0, 0, 0, 0, 0, 0]
  Call Extruder 0.09595
  MoveL (T745) to (118.95, 103.84, 1.1) mm, rotated rx 180 ry 0 rz -180 deg; joints [0, 0, 0, 0, 0, 0]
  Call Extruder 0.01786
  MoveL (T746) to (118.37, 103.84, 1.1) mm, rotated rx 180 ry 0 rz -180 deg; joints [0, 0, 0, 0, 0, 0]
  Call Extruder 0.12121
  MoveL (T747) to (121.16, 106.63, 1.1) mm, rotated rx 180 ry 0 rz -180 deg; joints [0, 0, 0, 0, 0, 0]
  Call Extruder 0.01786
  MoveL (T748) to (121.16, 107.21, 1.1) mm, rotated rx 180 ry 0 rz -180 deg; joints [0, 0, 0, 0, 0, 0]
  Call Extruder 0.14646
  MoveL (T749) to (117.79, 103.84, 1.1) mm, rotated rx 180 ry 0 rz -180 deg; joints [0, 0, 0, 0, 0, 0]
  Call Extruder 0.01786
  MoveL (T750) to (117.21, 103.84, 1.1) mm, rotated rx 180 ry 0 rz -180 deg; joints [0, 0, 0, 0, 0, 0]
  Call Extruder 0.17172
  MoveL (T751) to (121.16, 107.79, 1.1) mm, rotated rx 180 ry 0 rz -180 deg; joints [0, 0, 0, 0, 0, 0]
  Call Extruder 0.01786
  MoveL (T752) to (121.16, 108.38, 1.1) mm, rotated rx 180 ry 0 rz -180 deg; joints [0, 0, 0, 0, 0, 0]
  Call Extruder 0.19697
  MoveL (T753) to (116.62, 103.84, 1.1) mm, rotated rx 180 ry 0 rz -180 deg; joints [0, 0, 0, 0, 0, 0]
  Call Extruder 0.01786
  MoveL (T754) to (116.04, 103.84, 1.1) mm, rotated rx 180 ry 0 rz -180 deg; joints [0, 0, 0, 0, 0, 0]
  Call Extruder 0.22223
  MoveL (T755) to (121.16, 108.96, 1.1) mm, rotated rx 180 ry 0 rz -180 deg; joints [0, 0, 0, 0, 0, 0]
  Call Extruder 0.01786
  MoveL (T756) to (121.16, 109.54, 1.1) mm, rotated rx 180 ry 0 rz -180 deg; joints [0, 0, 0, 0, 0, 0]
